LIN {X 0,Y 248.2,Z 586.565,A -85,B 0,C 180,E1 -18983.497,E2 -18983.497} C_VEL
LIN {X 0,Y 249.035,Z 580.902,A -85,B 0,C 180,E1 -18985.954,E2 -18985.954} C_VEL
LIN {X 0,Y 250.181,Z 573.816,A -85,B 0,C 180,E1 -18988.39,E2 -18988.39} C_VEL
LIN {X 0,Y 251.663,Z 564.939,A -85,B 0,C 180,E1 -18990.8,E2 -18990.8} C_VEL
LIN {X 0,Y 253.35,Z 554.938,A -85,B 0,C 180,E1 -18992.961,E2 -18992.961} C_VEL
LIN {X 0,Y 254.867,Z 544.511,A -85,B 0,C 180,E1 -18994.745,E2 -18994.745} C_VEL
LIN {X 0,Y 256.41,Z 533.043,A -85,B 0,C 180,E1 -18996.294,E2 -18996.294} C_VEL
LIN {X 0,Y 257.735,Z 521.099,A -85,B 0,C 180,E1 -18997.54,E2 -18997.54} C_VEL
LIN {X 0,Y 258.808,Z 507.869,A -85,B 0,C 180,E1 -18998.54,E2 -18998.54} C_VEL
LIN {X 0,Y 259.542,Z 494.726,A -85,B 0,C 180,E1 -18999.203,E2 -18999.203} C_VEL
LIN {X 0,Y 261.752,Z 423.09,A -85,B 0,C 180,E1 -19001.164,E2 -19001.164} C_VEL
LIN {X 0,Y 256.331,Z 407.243,A -85,B 0,C 180,E1 -19002.139,E2 -19002.139} C_VEL
LIN {X 0,Y 251.283,Z 395.565,A -85,B 0,C 180,E1 -19002.996,E2 -19002.996} C_VEL
LIN {X 0,Y 249.318,Z 390.908,A -85,B 0,C 180,E1 -19003.344,E2 -19003.344} C_VEL
LIN {X 0,Y 249.246,Z 390.443,A -85,B 0,C 180,E1 -19003.4,E2 -19003.4} C_VEL
LIN {X 0,Y 249.222,Z 390.442,A -85,B 0,C 180,E1 -19006.503,E2 -19006.503} C_VEL
LIN {X 0,Y 249.091,Z 390.458,A -85,B 0,C 180,E1 -19011.517,E2 -19011.517} C_VEL
LIN {X 0,Y 249.134,Z 390.45,A -85,B 0,C 180,E1 -19015.481,E2 -19015.481} C_VEL
LIN {X 0,Y 249.086,Z 390.458,A -85,B 0,C 180,E1 -19018.992,E2 -19018.992} C_VEL
LIN {X 0,Y 249.032,Z 390.462,A -85,B 0,C 180,E1 -19022.425,E2 -19022.425} C_VEL
LIN {X 0,Y 249.031,Z 390.461,A -85,B 0,C 180,E1 -19026.344,E2 -19026.344} C_VEL
LIN {X 0,Y 249.006,Z 390.465,A -85,B 0,C 180,E1 -19030.477,E2 -19030.477} C_VEL
LIN {X 0,Y 249.007,Z 390.468,A -85,B 0,C 180,E1 -19034.877,E2 -19034.877} C_VEL
LIN {X 0,Y 249.017,Z 390.463,A -85,B 0,C 180,E1 -19037.362,E2 -19037.362} C_VEL
LIN {X 0,Y 249.041,Z 390.458,A -85,B 0,C 180,E1 -19042.199,E2 -19042.199} C_VEL
LIN {X 0,Y 249.041,Z 390.462,A -85,B 0,C 180,E1 -19045.638,E2 -19045.638} C_VEL
LIN {X 0,Y 249.049,Z 390.456,A -85,B 0,C 180,E1 -19049.472,E2 -19049.472} C_VEL
LIN {X 0,Y 249.07,Z 390.459,A -85,B 0,C 180,E1 -19053.161,E2 -19053.161} C_VEL
LIN {X 0,Y 249.076,Z 390.454,A -85,B 0,C 180,E1 -19056.732,E2 -19056.732} C_VEL
LIN {X 0,Y 249.107,Z 390.453,A -85,B 0,C 180,E1 -19060.211,E2 -19060.211} C_VEL
LIN {X 0,Y 249.238,Z 390.43,A -85,B 0,C 180,E1 -19063.621,E2 -19063.621} C_VEL
LIN {X 0,Y 249.24,Z 390.437,A -85,B 0,C 180,E1 -19068.615,E2 -19068.615} C_VEL
LIN {X 0,Y 249.449,Z 390.406,A -85,B 0,C 180,E1 -19071.901,E2 -19071.901} C_VEL
LIN {X 0,Y 249.292,Z 390.429,A -85,B 0,C 180,E1 -19075.148,E2 -19075.148} C_VEL
LIN {X 0,Y 249.67,Z 390.375,A -85,B 0,C 180,E1 -19078.387,E2 -19078.387} C_VEL
LIN {X 0,Y 249.671,Z 390.358,A -85,B 0,C 180,E1 -19081.613,E2 -19081.613} C_VEL
LIN {X 0,Y 249.448,Z 390.411,A -85,B 0,C 180,E1 -19086.47,E2 -19086.47} C_VEL
LIN {X 0,Y 249.308,Z 390.425,A -85,B 0,C 180,E1 -19090.006,E2 -19090.006} C_VEL
LIN {X 0,Y 248.561,Z 390.517,A -85,B 0,C 180,E1 -19091.353,E2 -19091.353} C_VEL
LIN {X 0,Y 245.711,Z 390.875,A -85,B 0,C 180,E1 -19093.55,E2 -19093.55} C_VEL
LIN {X 0,Y 242.481,Z 391.281,A -85,B 0,C 180,E1 -19096.256,E2 -19096.256} C_VEL
LIN {X 0,Y 242.115,Z 391.32,A -85,B 0,C 180,E1 -19097.193,E2 -19097.193} C_VEL
LIN {X 0,Y 242.008,Z 391.34,A -85,B 0,C 180,E1 -19102.18,E2 -19102.18} C_VEL
LIN {X 0,Y 242.062,Z 391.333,A -85,B 0,C 180,E1 -19105.838,E2 -19105.838} C_VEL
LIN {X 0,Y 242.027,Z 391.337,A -85,B 0,C 180,E1 -19109.58,E2 -19109.58} C_VEL
LIN {X 0,Y 241.988,Z 391.343,A -85,B 0,C 180,E1 -19113.491,E2 -19113.491} C_VEL
LIN {X 0,Y 242.009,Z 391.342,A -85,B 0,C 180,E1 -19117.578,E2 -19117.578} C_VEL
LIN {X 0,Y 241.982,Z 391.348,A -85,B 0,C 180,E1 -19121.913,E2 -19121.913} C_VEL
LIN {X 0,Y 241.983,Z 391.344,A -85,B 0,C 180,E1 -19126.559,E2 -19126.559} C_VEL
LIN {X 0,Y 241.986,Z 391.339,A -85,B 0,C 180,E1 -19130.288,E2 -19130.288} C_VEL
LIN {X 0,Y 242.097,Z 391.377,A -85,B 0,C 180,E1 -19133.66,E2 -19133.66} C_VEL
LIN {X 0,Y 244.057,Z 400.843,A -85,B 0,C 180,E1 -19137.322,E2 -19137.322} C_VEL
LIN {X 0,Y 245.642,Z 408.584,A -85,B 0,C 180,E1 -19140.173,E2 -19140.173} C_VEL
LIN {X 0,Y 249.345,Z 419.538,A -85,B 0,C 180,E1 -19140.898,E2 -19140.898} C_VEL
LIN {X 0,Y 254.277,Z 461.944,A -85,B 0,C 180,E1 -19142.67,E2 -19142.67} C_VEL
LIN {X 0,Y 252.511,Z 517.102,A -85,B 0,C 180,E1 -19144.223,E2 -19144.223} C_VEL
LIN {X 0,Y 251.666,Z 530.452,A -85,B 0,C 180,E1 -19144.905,E2 -19144.905} C_VEL
LIN {X 0,Y 250.342,Z 543.226,A -85,B 0,C 180,E1 -19145.87,E2 -19145.87} C_VEL
LIN {X 0,Y 248.767,Z 555.378,A -85,B 0,C 180,E1 -19147.142,E2 -19147.142} C_VEL
LIN {X 0,Y 247.124,Z 565.64,A -85,B 0,C 180,E1 -19148.522,E2 -19148.522} C_VEL
LIN {X 0,Y 245.467,Z 576.326,A -85,B 0,C 180,E1 -19150.342,E2 -19150.342} C_VEL
LIN {X 0,Y 243.996,Z 584.587,A -85,B 0,C 180,E1 -19152.074,E2 -19152.074} C_VEL
LIN {X 0,Y 243.116,Z 590.805,A -85,B 0,C 180,E1 -19153.63,E2 -19153.63} C_VEL
LIN {X 0,Y 241.774,Z 599.073,A -85,B 0,C 180,E1 -19156.125,E2 -19156.125} C_VEL
LIN {X 0,Y 240.907,Z 604.686,A -85,B 0,C 180,E1 -19158.217,E2 -19158.217} C_VEL
LIN {X 0,Y 240.332,Z 610.169,A -85,B 0,C 180,E1 -19160.745,E2 -19160.745} C_VEL
LIN {X 0,Y 240.044,Z 614.433,A -85,B 0,C 180,E1 -19163.275,E2 -19163.275} C_VEL
LIN {X 0,Y 239.922,Z 616.68,A -85,B 0,C 180,E1 -19164.959,E2 -19164.959} C_VEL
LIN {X 0,Y 239.977,Z 618.439,A -85,B 0,C 180,E1 -19166.642,E2 -19166.642} C_VEL
LIN {X 0,Y 240.01,Z 619.761,A -85,B 0,C 180,E1 -19168.322,E2 -19168.322} C_VEL
LIN {X 0,Y 240.022,Z 620.676,A -85,B 0,C 180,E1 -19170,E2 -19170} C_VEL
LIN {X 0,Y 239.976,Z 621.188,A -85,B 0,C 180,E1 -19171.678,E2 -19171.678} C_VEL
LIN {X 0,Y 239.911,Z 621.261,A -85,B 0,C 180,E1 -19173.359,E2 -19173.359} C_VEL
LIN {X 0,Y 239.912,Z 620.913,A -85,B 0,C 180,E1 -19175.127,E2 -19175.127} C_VEL
LIN {X 0,Y 240.163,Z 619.15,A -85,B 0,C 180,E1 -19178.413,E2 -19178.413} C_VEL
LIN {X 0,Y 240.571,Z 617.639,A -85,B 0,C 180,E1 -19180.095,E2 -19180.095} C_VEL
LIN {X 0,Y 241.434,Z 614.593,A -85,B 0,C 180,E1 -19182.61,E2 -19182.61} C_VEL
LIN {X 0,Y 242.852,Z 610.525,A -85,B 0,C 180,E1 -19185.097,E2 -19185.097} C_VEL
LIN {X 0,Y 245.038,Z 604.321,A -85,B 0,C 180,E1 -19187.958,E2 -19187.958} C_VEL
LIN {X 0,Y 247.264,Z 597.853,A -85,B 0,C 180,E1 -19190.288,E2 -19190.288} C_VEL
LIN {X 0,Y 250.083,Z 589.313,A -85,B 0,C 180,E1 -19192.731,E2 -19192.731} C_VEL
LIN {X 0,Y 252.865,Z 580.828,A -85,B 0,C 180,E1 -19194.639,E2 -19194.639} C_VEL
LIN {X 0,Y 255.921,Z 570.39,A -85,B 0,C 180,E1 -19196.503,E2 -19196.503} C_VEL
LIN {X 0,Y 258.611,Z 560.094,A -85,B 0,C 180,E1 -19197.955,E2 -19197.955} C_VEL
LIN {X 0,Y 261.177,Z 548.836,A -85,B 0,C 180,E1 -19199.19,E2 -19199.19} C_VEL
LIN {X 0,Y 263.441,Z 536.133,A -85,B 0,C 180,E1 -19200.234,E2 -19200.234} C_VEL
LIN {X 0,Y 265.184,Z 522.682,A -85,B 0,C 180,E1 -19201.001,E2 -19201.001} C_VEL
LIN {X 0,Y 266.181,Z 510.056,A -85,B 0,C 180,E1 -19201.448,E2 -19201.448} C_VEL
LIN {X 0,Y 268.042,Z 465.142,A -85,B 0,C 180,E1 -19202.66,E2 -19202.66} C_VEL
LIN {X 0,Y 265.308,Z 446.292,A -85,B 0,C 180,E1 -19203.775,E2 -19203.775} C_VEL
LIN {X 0,Y 264.329,Z 441.703,A -85,B 0,C 180,E1 -19204.109,E2 -19204.109} C_VEL
LIN {X 0,Y 256.778,Z 425.571,A -85,B 0,C 180,E1 -19206.11,E2 -19206.11} C_VEL
LIN {X 0,Y 250.954,Z 414.885,A -85,B 0,C 180,E1 -19207.723,E2 -19207.723} C_VEL
LIN {X 0,Y 248.498,Z 410.557,A -85,B 0,C 180,E1 -19208.435,E2 -19208.435} C_VEL
LIN {X 0,Y 246.306,Z 406.343,A -85,B 0,C 180,E1 -19209.128,E2 -19209.128} C_VEL
LIN {X 0,Y 244.316,Z 399.158,A -85,B 0,C 180,E1 -19212.818,E2 -19212.818} C_VEL
LIN {X 0,Y 242.033,Z 391.332,A -85,B 0,C 180,E1 -19217.362,E2 -19217.362} C_VEL
LIN {X 0,Y 242.016,Z 391.34,A -85,B 0,C 180,E1 -19221.632,E2 -19221.632} C_VEL
LIN {X 0,Y 242.033,Z 391.336,A -85,B 0,C 180,E1 -19224.497,E2 -19224.497} C_VEL
LIN {X 0,Y 241.973,Z 391.343,A -85,B 0,C 180,E1 -19228.48,E2 -19228.48} C_VEL
LIN {X 0,Y 242.007,Z 391.338,A -85,B 0,C 180,E1 -19232.313,E2 -19232.313} C_VEL
LIN {X 0,Y 242.053,Z 391.334,A -85,B 0,C 180,E1 -19236.016,E2 -19236.016} C_VEL
LIN {X 0,Y 242.033,Z 391.331,A -85,B 0,C 180,E1 -19239.608,E2 -19239.608} C_VEL
LIN {X 0,Y 242.159,Z 391.308,A -85,B 0,C 180,E1 -19243.278,E2 -19243.278} C_VEL
LIN {X 0,Y 242.18,Z 391.306,A -85,B 0,C 180,E1 -19248.28,E2 -19248.28} C_VEL
LIN {X 0,Y 242.421,Z 391.276,A -85,B 0,C 180,E1 -19251.666,E2 -19251.666} C_VEL
LIN {X 0,Y 242.255,Z 391.309,A -85,B 0,C 180,E1 -19255.007,E2 -19255.007} C_VEL
LIN {X 0,Y 242.631,Z 391.25,A -85,B 0,C 180,E1 -19258.341,E2 -19258.341} C_VEL
LIN {X 0,Y 242.632,Z 391.25,A -85,B 0,C 180,E1 -19261.66,E2 -19261.66} C_VEL
LIN {X 0,Y 242.417,Z 391.277,A -85,B 0,C 180,E1 -19266.684,E2 -19266.684} C_VEL
LIN {X 0,Y 242.263,Z 391.308,A -85,B 0,C 180,E1 -19270.024,E2 -19270.024} C_VEL
LIN {X 0,Y 242.16,Z 391.315,A -85,B 0,C 180,E1 -19275.142,E2 -19275.142} C_VEL
LIN {X 0,Y 242.085,Z 391.331,A -85,B 0,C 180,E1 -19278.624,E2 -19278.624} C_VEL
LIN {X 0,Y 242.06,Z 391.334,A -85,B 0,C 180,E1 -19282.176,E2 -19282.176} C_VEL
LIN {X 0,Y 242.064,Z 391.333,A -85,B 0,C 180,E1 -19285.839,E2 -19285.839} C_VEL
LIN {X 0,Y 242.028,Z 391.335,A -85,B 0,C 180,E1 -19289.581,E2 -19289.581} C_VEL
LIN {X 0,Y 242.006,Z 391.394,A -85,B 0,C 180,E1 -19293.927,E2 -19293.927} C_VEL
LIN {X 0,Y 242.958,Z 394.034,A -85,B 0,C 180,E1 -19294.276,E2 -19294.276} C_VEL
LIN {X 0,Y 245.31,Z 396.811,A -85,B 0,C 180,E1 -19294.96,E2 -19294.96} C_VEL
LIN {X 0,Y 247.486,Z 400.114,A -85,B 0,C 180,E1 -19295.603,E2 -19295.603} C_VEL
LIN {X 0,Y 252.215,Z 407.1,A -85,B 0,C 180,E1 -19296.931,E2 -19296.931} C_VEL
LIN {X 0,Y 256.167,Z 413.341,A -85,B 0,C 180,E1 -19297.995,E2 -19297.995} C_VEL
LIN {X 0,Y 262.545,Z 425.008,A -85,B 0,C 180,E1 -19299.663,E2 -19299.663} C_VEL
LIN {X 0,Y 269.196,Z 439.033,A -85,B 0,C 180,E1 -19301.334,E2 -19301.334} C_VEL
LIN {X 0,Y 266.535,Z 496.566,A -85,B 0,C 180,E1 -19302.897,E2 -19302.897} C_VEL
LIN {X 0,Y 265.248,Z 510.053,A -85,B 0,C 180,E1 -19303.557,E2 -19303.557} C_VEL
LIN {X 0,Y 263.535,Z 522.714,A -85,B 0,C 180,E1 -19304.491,E2 -19304.491} C_VEL
LIN {X 0,Y 261.43,Z 534.297,A -85,B 0,C 180,E1 -19305.658,E2 -19305.658} C_VEL
LIN {X 0,Y 258.738,Z 546.27,A -85,B 0,C 180,E1 -19307.231,E2 -19307.231} C_VEL
LIN {X 0,Y 255.936,Z 556.885,A -85,B 0,C 180,E1 -19309.035,E2 -19309.035} C_VEL
LIN {X 0,Y 253.085,Z 566.205,A -85,B 0,C 180,E1 -19311.037,E2 -19311.037} C_VEL
LIN {X 0,Y 250.205,Z 574.762,A -85,B 0,C 180,E1 -19313.354,E2 -19313.354} C_VEL
LIN {X 0,Y 247.553,Z 582.051,A -85,B 0,C 180,E1 -19315.897,E2 -19315.897} C_VEL
LIN {X 0,Y 245.653,Z 586.942,A -85,B 0,C 180,E1 -19318.044,E2 -19318.044} C_VEL
LIN {X 0,Y 243.746,Z 591.546,A -85,B 0,C 180,E1 -19320.649,E2 -19320.649} C_VEL
LIN {X 0,Y 242.75,Z 593.944,A -85,B 0,C 180,E1 -19322.405,E2 -19322.405} C_VEL
LIN {X 0,Y 241.831,Z 595.977,A -85,B 0,C 180,E1 -19324.28,E2 -19324.28} C_VEL
LIN {X 0,Y 241.168,Z 597.278,A -85,B 0,C 180,E1 -19325.923,E2 -19325.923} C_VEL
LIN {X 0,Y 240.612,Z 598.253,A -85,B 0,C 180,E1 -19327.685,E2 -19327.685} C_VEL
LIN {X 0,Y 240.229,Z 598.811,A -85,B 0,C 180,E1 -19329.448,E2 -19329.448} C_VEL
LIN {X 0,Y 239.924,Z 598.91,A -85,B 0,C 180,E1 -19331.203,E2 -19331.203} C_VEL
LIN {X 0,Y 239.738,Z 598.584,A -85,B 0,C 180,E1 -19332.954,E2 -19332.954} C_VEL
LIN {X 0,Y 239.758,Z 597.487,A -85,B 0,C 180,E1 -19335.316,E2 -19335.316} C_VEL
LIN {X 0,Y 239.919,Z 595.083,A -85,B 0,C 180,E1 -19338.168,E2 -19338.168} C_VEL
LIN {X 0,Y 240.385,Z 591.842,A -85,B 0,C 180,E1 -19340.747,E2 -19340.747} C_VEL
LIN {X 0,Y 241.044,Z 587.519,A -85,B 0,C 180,E1 -19343.303,E2 -19343.303} C_VEL
LIN {X 0,Y 242.05,Z 580.982,A -85,B 0,C 180,E1 -19346.254,E2 -19346.254} C_VEL
LIN {X 0,Y 243.251,Z 573.809,A -85,B 0,C 180,E1 -19348.758,E2 -19348.758} C_VEL
LIN {X 0,Y 244.805,Z 564.86,A -85,B 0,C 180,E1 -19351.234,E2 -19351.234} C_VEL
LIN {X 0,Y 246.404,Z 555.67,A -85,B 0,C 180,E1 -19353.27,E2 -19353.27} C_VEL
LIN {X 0,Y 247.956,Z 545.486,A -85,B 0,C 180,E1 -19355.081,E2 -19355.081} C_VEL
LIN {X 0,Y 249.542,Z 534.158,A -85,B 0,C 180,E1 -19356.671,E2 -19356.671} C_VEL
LIN {X 0,Y 250.906,Z 522.441,A -85,B 0,C 180,E1 -19357.949,E2 -19357.949} C_VEL
LIN {X 0,Y 252.022,Z 509.688,A -85,B 0,C 180,E1 -19358.974,E2 -19358.974} C_VEL
LIN {X 0,Y 252.832,Z 496.157,A -85,B 0,C 180,E1 -19359.701,E2 -19359.701} C_VEL
LIN {X 0,Y 254.305,Z 452.666,A -85,B 0,C 180,E1 -19360.949,E2 -19360.949} C_VEL
LIN {X 0,Y 255.146,Z 424.433,A -85,B 0,C 180,E1 -19361.729,E2 -19361.729} C_VEL
LIN {X 0,Y 249.638,Z 408.47,A -85,B 0,C 180,E1 -19362.759,E2 -19362.759} C_VEL
LIN {X 0,Y 242.958,Z 393.784,A -85,B 0,C 180,E1 -19363.926,E2 -19363.926} C_VEL
LIN {X 0,Y 242.189,Z 391.321,A -85,B 0,C 180,E1 -19364.14,E2 -19364.14} C_VEL
LIN {X 0,Y 242.154,Z 391.324,A -85,B 0,C 180,E1 -19366.871,E2 -19366.871} C_VEL
LIN {X 0,Y 242.056,Z 391.333,A -85,B 0,C 180,E1 -19371.702,E2 -19371.702} C_VEL
LIN {X 0,Y 242.069,Z 391.332,A -85,B 0,C 180,E1 -19375.837,E2 -19375.837} C_VEL
LIN {X 0,Y 242.032,Z 391.338,A -85,B 0,C 180,E1 -19379.579,E2 -19379.579} C_VEL
LIN {X 0,Y 241.982,Z 391.344,A -85,B 0,C 180,E1 -19383.491,E2 -19383.491} C_VEL
LIN {X 0,Y 241.988,Z 391.34,A -85,B 0,C 180,E1 -19387.581,E2 -19387.581} C_VEL
LIN {X 0,Y 241.939,Z 391.342,A -85,B 0,C 180,E1 -19391.921,E2 -19391.921} C_VEL
LIN {X 0,Y 241.936,Z 391.344,A -85,B 0,C 180,E1 -19396.569,E2 -19396.569} C_VEL
LIN {X 0,Y 241.955,Z 391.344,A -85,B 0,C 180,E1 -19400.28,E2 -19400.28} C_VEL
LIN {X 0,Y 241.979,Z 391.34,A -85,B 0,C 180,E1 -19404.487,E2 -19404.487} C_VEL
LIN {X 0,Y 241.972,Z 391.342,A -85,B 0,C 180,E1 -19408.479,E2 -19408.479} C_VEL
LIN {X 0,Y 242.005,Z 391.338,A -85,B 0,C 180,E1 -19412.312,E2 -19412.312} C_VEL
LIN {X 0,Y 242.054,Z 391.327,A -85,B 0,C 180,E1 -19416.015,E2 -19416.015} C_VEL
LIN {X 0,Y 242.034,Z 391.334,A -85,B 0,C 180,E1 -19419.607,E2 -19419.607} C_VEL
LIN {X 0,Y 242.16,Z 391.312,A -85,B 0,C 180,E1 -19423.277,E2 -19423.277} C_VEL
LIN {X 0,Y 242.176,Z 391.317,A -85,B 0,C 180,E1 -19428.279,E2 -19428.279} C_VEL
LIN {X 0,Y 242.395,Z 391.284,A -85,B 0,C 180,E1 -19431.664,E2 -19431.664} C_VEL
LIN {X 0,Y 242.253,Z 391.306,A -85,B 0,C 180,E1 -19435.007,E2 -19435.007} C_VEL
LIN {X 0,Y 242.631,Z 391.251,A -85,B 0,C 180,E1 -19438.34,E2 -19438.34} C_VEL
LIN {X 0,Y 242.631,Z 391.233,A -85,B 0,C 180,E1 -19441.659,E2 -19441.659} C_VEL
LIN {X 0,Y 242.418,Z 391.288,A -85,B 0,C 180,E1 -19446.659,E2 -19446.659} C_VEL
LIN {X 0,Y 242.262,Z 391.307,A -85,B 0,C 180,E1 -19450.024,E2 -19450.024} C_VEL
LIN {X 0,Y 242.159,Z 391.319,A -85,B 0,C 180,E1 -19455.141,E2 -19455.141} C_VEL
LIN {X 0,Y 242.115,Z 391.32,A -85,B 0,C 180,E1 -19457.193,E2 -19457.193} C_VEL
LIN {X 0,Y 241.351,Z 391.419,A -85,B 0,C 180,E1 -19458.582,E2 -19458.582} C_VEL
LIN {X 0,Y 238.408,Z 391.787,A -85,B 0,C 180,E1 -19460.845,E2 -19460.845} C_VEL
LIN {X 0,Y 235.996,Z 392.085,A -85,B 0,C 180,E1 -19462.691,E2 -19462.691} C_VEL
LIN {X 0,Y 235.022,Z 392.207,A -85,B 0,C 180,E1 -19464.123,E2 -19464.123} C_VEL
LIN {X 0,Y 234.972,Z 392.214,A -85,B 0,C 180,E1 -19464.608,E2 -19464.608} C_VEL
LIN {X 0,Y 234.95,Z 392.219,A -85,B 0,C 180,E1 -19468.594,E2 -19468.594} C_VEL
LIN {X 0,Y 234.946,Z 392.22,A -85,B 0,C 180,E1 -19473.118,E2 -19473.118} C_VEL
LIN {X 0,Y 234.943,Z 392.222,A -85,B 0,C 180,E1 -19476.746,E2 -19476.746} C_VEL
LIN {X 0,Y 234.942,Z 392.223,A -85,B 0,C 180,E1 -19481.155,E2 -19481.155} C_VEL
LIN {X 0,Y 234.939,Z 392.224,A -85,B 0,C 180,E1 -19484.117,E2 -19484.117} C_VEL
LIN {X 0,Y 234.939,Z 392.22,A -85,B 0,C 180,E1 -19488.405,E2 -19488.405} C_VEL
LIN {X 0,Y 235.035,Z 392.347,A -85,B 0,C 180,E1 -19493.138,E2 -19493.138} C_VEL
LIN {X 0,Y 237.018,Z 401.538,A -85,B 0,C 180,E1 -19496.831,E2 -19496.831} C_VEL
LIN {X 0,Y 238.366,Z 408.281,A -85,B 0,C 180,E1 -19499.385,E2 -19499.385} C_VEL
LIN {X 0,Y 242.902,Z 420.907,A -85,B 0,C 180,E1 -19500.283,E2 -19500.283} C_VEL
LIN {X 0,Y 247.686,Z 462.997,A -85,B 0,C 180,E1 -19502.096,E2 -19502.096} C_VEL
LIN {X 0,Y 245.866,Z 516.715,A -85,B 0,C 180,E1 -19503.644,E2 -19503.644} C_VEL
LIN {X 0,Y 245.002,Z 530.089,A -85,B 0,C 180,E1 -19504.344,E2 -19504.344} C_VEL
LIN {X 0,Y 243.565,Z 543.426,A -85,B 0,C 180,E1 -19505.381,E2 -19505.381} C_VEL
LIN {X 0,Y 241.956,Z 555.431,A -85,B 0,C 180,E1 -19506.687,E2 -19506.687} C_VEL
LIN {X 0,Y 240.268,Z 565.623,A -85,B 0,C 180,E1 -19508.103,E2 -19508.103} C_VEL
LIN {X 0,Y 238.559,Z 576.255,A -85,B 0,C 180,E1 -19509.973,E2 -19509.973} C_VEL
LIN {X 0,Y 236.855,Z 586.018,A -85,B 0,C 180,E1 -19512.128,E2 -19512.128} C_VEL
LIN {X 0,Y 235.461,Z 594.309,A -85,B 0,C 180,E1 -19514.418,E2 -19514.418} C_VEL
LIN {X 0,Y 234.218,Z 601.815,A -85,B 0,C 180,E1 -19516.995,E2 -19516.995} C_VEL
LIN {X 0,Y 233.46,Z 607.834,A -85,B 0,C 180,E1 -19519.594,E2 -19519.594} C_VEL
LIN {X 0,Y 233.047,Z 612.567,A -85,B 0,C 180,E1 -19522.201,E2 -19522.201} C_VEL
LIN {X 0,Y 232.845,Z 616.267,A -85,B 0,C 180,E1 -19524.9,E2 -19524.9} C_VEL
LIN {X 0,Y 232.891,Z 617.97,A -85,B 0,C 180,E1 -19526.54,E2 -19526.54} C_VEL
LIN {X 0,Y 232.939,Z 619.324,A -85,B 0,C 180,E1 -19528.271,E2 -19528.271} C_VEL
LIN {X 0,Y 232.95,Z 620.268,A -85,B 0,C 180,E1 -19530,E2 -19530} C_VEL
LIN {X 0,Y 232.905,Z 620.812,A -85,B 0,C 180,E1 -19531.729,E2 -19531.729} C_VEL
LIN {X 0,Y 232.801,Z 620.715,A -85,B 0,C 180,E1 -19534.976,E2 -19534.976} C_VEL
LIN {X 0,Y 232.883,Z 619.974,A -85,B 0,C 180,E1 -19536.933,E2 -19536.933} C_VEL
LIN {X 0,Y 233.549,Z 617.467,A -85,B 0,C 180,E1 -19540.402,E2 -19540.402} C_VEL
LIN {X 0,Y 234.457,Z 614.472,A -85,B 0,C 180,E1 -19542.992,E2 -19542.992} C_VEL
LIN {X 0,Y 235.982,Z 610.466,A -85,B 0,C 180,E1 -19545.547,E2 -19545.547} C_VEL
LIN {X 0,Y 238.274,Z 604.363,A -85,B 0,C 180,E1 -19548.486,E2 -19548.486} C_VEL
LIN {X 0,Y 240.466,Z 598.409,A -85,B 0,C 180,E1 -19550.732,E2 -19550.732} C_VEL
LIN {X 0,Y 243.036,Z 591.024,A -85,B 0,C 180,E1 -19552.978,E2 -19552.978} C_VEL
LIN {X 0,Y 245.818,Z 582.974,A -85,B 0,C 180,E1 -19554.942,E2 -19554.942} C_VEL
LIN {X 0,Y 248.948,Z 573.186,A -85,B 0,C 180,E1 -19556.852,E2 -19556.852} C_VEL
LIN {X 0,Y 252.025,Z 562.289,A -85,B 0,C 180,E1 -19558.525,E2 -19558.525} C_VEL
LIN {X 0,Y 255.055,Z 549.886,A -85,B 0,C 180,E1 -19559.962,E2 -19559.962} C_VEL
LIN {X 0,Y 257.392,Z 537.756,A -85,B 0,C 180,E1 -19561.022,E2 -19561.022} C_VEL
LIN {X 0,Y 259.221,Z 525.047,A -85,B 0,C 180,E1 -19561.805,E2 -19561.805} C_VEL
LIN {X 0,Y 260.368,Z 512.937,A -85,B 0,C 180,E1 -19562.289,E2 -19562.289} C_VEL
LIN {X 0,Y 262.443,Z 466.155,A -85,B 0,C 180,E1 -19563.584,E2 -19563.584} C_VEL
LIN {X 0,Y 259.786,Z 447.749,A -85,B 0,C 180,E1 -19564.719,E2 -19564.719} C_VEL
LIN {X 0,Y 258.954,Z 444.374,A -85,B 0,C 180,E1 -19564.996,E2 -19564.996} C_VEL
LIN {X 0,Y 251.979,Z 429.485,A -85,B 0,C 180,E1 -19566.938,E2 -19566.938} C_VEL
LIN {X 0,Y 246.41,Z 418.994,A -85,B 0,C 180,E1 -19568.562,E2 -19568.562} C_VEL
LIN {X 0,Y 241.671,Z 410.659,A -85,B 0,C 180,E1 -19570.019,E2 -19570.019} C_VEL
LIN {X 0,Y 239.166,Z 406.342,A -85,B 0,C 180,E1 -19570.827,E2 -19570.827} C_VEL
LIN {X 0,Y 238.913,Z 405.628,A -85,B 0,C 180,E1 -19571.033,E2 -19571.033} C_VEL
LIN {X 0,Y 237.013,Z 399.189,A -85,B 0,C 180,E1 -19574.63,E2 -19574.63} C_VEL
LIN {X 0,Y 234.975,Z 392.217,A -85,B 0,C 180,E1 -19578.994,E2 -19578.994} C_VEL
LIN {X 0,Y 234.943,Z 392.212,A -85,B 0,C 180,E1 -19583.254,E2 -19583.254} C_VEL
LIN {X 0,Y 234.956,Z 392.212,A -85,B 0,C 180,E1 -19587.424,E2 -19587.424} C_VEL
LIN {X 0,Y 234.95,Z 392.215,A -85,B 0,C 180,E1 -19591.406,E2 -19591.406} C_VEL
LIN {X 0,Y 234.983,Z 392.209,A -85,B 0,C 180,E1 -19595.246,E2 -19595.246} C_VEL
LIN {X 0,Y 235.007,Z 392.201,A -85,B 0,C 180,E1 -19598.97,E2 -19598.97} C_VEL
LIN {X 0,Y 235.091,Z 392.187,A -85,B 0,C 180,E1 -19603.06,E2 -19603.06} C_VEL
LIN {X 0,Y 235.112,Z 392.185,A -85,B 0,C 180,E1 -19607.922,E2 -19607.922} C_VEL
LIN {X 0,Y 235.371,Z 392.156,A -85,B 0,C 180,E1 -19611.414,E2 -19611.414} C_VEL
LIN {X 0,Y 235.397,Z 392.148,A -85,B 0,C 180,E1 -19613.142,E2 -19613.142} C_VEL
LIN {X 0,Y 235.591,Z 392.126,A -85,B 0,C 180,E1 -19618.291,E2 -19618.291} C_VEL
LIN {X 0,Y 235.591,Z 392.126,A -85,B 0,C 180,E1 -19621.71,E2 -19621.71} C_VEL
LIN {X 0,Y 235.369,Z 392.154,A -85,B 0,C 180,E1 -19626.86,E2 -19626.86} C_VEL
LIN {X 0,Y 235.21,Z 392.185,A -85,B 0,C 180,E1 -19630.328,E2 -19630.328} C_VEL
LIN {X 0,Y 235.108,Z 392.189,A -85,B 0,C 180,E1 -19635.607,E2 -19635.607} C_VEL
LIN {X 0,Y 235.025,Z 392.205,A -85,B 0,C 180,E1 -19639.205,E2 -19639.205} C_VEL
LIN {X 0,Y 234.986,Z 392.21,A -85,B 0,C 180,E1 -19642.881,E2 -19642.881} C_VEL
LIN {X 0,Y 234.967,Z 392.212,A -85,B 0,C 180,E1 -19646.658,E2 -19646.658} C_VEL
LIN {X 0,Y 234.93,Z 392.216,A -85,B 0,C 180,E1 -19650.569,E2 -19650.569} C_VEL
LIN {X 0,Y 234.946,Z 392.219,A -85,B 0,C 180,E1 -19652.071,E2 -19652.071} C_VEL
LIN {X 0,Y 235.961,Z 395.087,A -85,B 0,C 180,E1 -19652.517,E2 -19652.517} C_VEL
LIN {X 0,Y 238.394,Z 397.754,A -85,B 0,C 180,E1 -19653.283,E2 -19653.283} C_VEL
LIN {X 0,Y 240.524,Z 401.042,A -85,B 0,C 180,E1 -19653.971,E2 -19653.971} C_VEL
LIN {X 0,Y 241.984,Z 402.995,A -85,B 0,C 180,E1 -19654.417,E2 -19654.417} C_VEL
LIN {X 0,Y 247.628,Z 411.237,A -85,B 0,C 180,E1 -19656.088,E2 -19656.088} C_VEL
LIN {X 0,Y 252.19,Z 418.616,A -85,B 0,C 180,E1 -19657.373,E2 -19657.373} C_VEL
LIN {X 0,Y 258.595,Z 430.57,A -85,B 0,C 180,E1 -19659.119,E2 -19659.119} C_VEL
LIN {X 0,Y 263.574,Z 441.238,A -85,B 0,C 180,E1 -19660.428,E2 -19660.428} C_VEL
LIN {X 0,Y 260.928,Z 496.621,A -85,B 0,C 180,E1 -19661.958,E2 -19661.958} C_VEL
LIN {X 0,Y 259.625,Z 509.957,A -85,B 0,C 180,E1 -19662.614,E2 -19662.614} C_VEL
LIN {X 0,Y 257.941,Z 522.004,A -85,B 0,C 180,E1 -19663.496,E2 -19663.496} C_VEL
LIN {X 0,Y 255.734,Z 533.877,A -85,B 0,C 180,E1 -19664.678,E2 -19664.678} C_VEL
LIN {X 0,Y 253.056,Z 545.623,A -85,B 0,C 180,E1 -19666.228,E2 -19666.228} C_VEL
LIN {X 0,Y 250.301,Z 555.665,A -85,B 0,C 180,E1 -19667.906,E2 -19667.906} C_VEL
LIN {X 0,Y 247.333,Z 565.115,A -85,B 0,C 180,E1 -19669.897,E2 -19669.897} C_VEL
LIN {X 0,Y 244.2,Z 574.052,A -85,B 0,C 180,E1 -19672.298,E2 -19672.298} C_VEL
LIN {X 0,Y 241.277,Z 581.709,A -85,B 0,C 180,E1 -19674.934,E2 -19674.934} C_VEL
LIN {X 0,Y 239.284,Z 586.61,A -85,B 0,C 180,E1 -19677.088,E2 -19677.088} C_VEL
LIN {X 0,Y 237.219,Z 591.397,A -85,B 0,C 180,E1 -19679.759,E2 -19679.759} C_VEL
LIN {X 0,Y 235.593,Z 594.954,A -85,B 0,C 180,E1 -19682.46,E2 -19682.46} C_VEL
LIN {X 0,Y 234.344,Z 597.405,A -85,B 0,C 180,E1 -19685.175,E2 -19685.175} C_VEL
LIN {X 0,Y 233.719,Z 598.443,A -85,B 0,C 180,E1 -19686.989,E2 -19686.989} C_VEL
LIN {X 0,Y 233.218,Z 599.137,A -85,B 0,C 180,E1 -19689.098,E2 -19689.098} C_VEL
LIN {X 0,Y 232.704,Z 599.019,A -85,B 0,C 180,E1 -19692.422,E2 -19692.422} C_VEL
LIN {X 0,Y 232.661,Z 597.845,A -85,B 0,C 180,E1 -19695.159,E2 -19695.159} C_VEL
LIN {X 0,Y 232.797,Z 595.763,A -85,B 0,C 180,E1 -19697.8,E2 -19697.8} C_VEL
LIN {X 0,Y 233.228,Z 592.651,A -85,B 0,C 180,E1 -19700.46,E2 -19700.46} C_VEL
LIN {X 0,Y 233.881,Z 588.463,A -85,B 0,C 180,E1 -19703.097,E2 -19703.097} C_VEL
LIN {X 0,Y 234.895,Z 582.072,A -85,B 0,C 180,E1 -19706.14,E2 -19706.14} C_VEL
LIN {X 0,Y 236.112,Z 575.12,A -85,B 0,C 180,E1 -19708.721,E2 -19708.721} C_VEL
LIN {X 0,Y 237.661,Z 566.409,A -85,B 0,C 180,E1 -19711.271,E2 -19711.271} C_VEL
LIN {X 0,Y 239.411,Z 556.66,A -85,B 0,C 180,E1 -19713.537,E2 -19713.537} C_VEL
LIN {X 0,Y 241.055,Z 546.44,A -85,B 0,C 180,E1 -19715.437,E2 -19715.437} C_VEL
LIN {X 0,Y 242.683,Z 535.256,A -85,B 0,C 180,E1 -19717.07,E2 -19717.07} C_VEL
LIN {X 0,Y 244.209,Z 522.736,A -85,B 0,C 180,E1 -19718.481,E2 -19718.481} C_VEL
LIN {X 0,Y 245.351,Z 509.978,A -85,B 0,C 180,E1 -19719.532,E2 -19719.532} C_VEL
LIN {X 0,Y 246.213,Z 496.07,A -85,B 0,C 180,E1 -19720.292,E2 -19720.292} C_VEL
LIN {X 0,Y 248.548,Z 425.66,A -85,B 0,C 180,E1 -19722.329,E2 -19722.329} C_VEL
LIN {X 0,Y 243.034,Z 409.951,A -85,B 0,C 180,E1 -19723.395,E2 -19723.395} C_VEL
LIN {X 0,Y 235.305,Z 393.123,A -85,B 0,C 180,E1 -19724.806,E2 -19724.806} C_VEL
LIN {X 0,Y 235.14,Z 392.199,A -85,B 0,C 180,E1 -19724.879,E2 -19724.879} C_VEL
LIN {X 0,Y 235.013,Z 392.213,A -85,B 0,C 180,E1 -19729.205,E2 -19729.205} C_VEL
LIN {X 0,Y 234.964,Z 392.213,A -85,B 0,C 180,E1 -19732.882,E2 -19732.882} C_VEL
LIN {X 0,Y 234.973,Z 392.216,A -85,B 0,C 180,E1 -19736.656,E2 -19736.656} C_VEL
LIN {X 0,Y 234.934,Z 392.221,A -85,B 0,C 180,E1 -19740.567,E2 -19740.567} C_VEL
LIN {X 0,Y 234.928,Z 392.221,A -85,B 0,C 180,E1 -19744.637,E2 -19744.637} C_VEL
LIN {X 0,Y 234.942,Z 392.22,A -85,B 0,C 180,E1 -19748.943,E2 -19748.943} C_VEL
LIN {X 0,Y 234.889,Z 392.225,A -85,B 0,C 180,E1 -19753.484,E2 -19753.484} C_VEL
LIN {X 0,Y 234.889,Z 392.222,A -85,B 0,C 180,E1 -19756.513,E2 -19756.513} C_VEL
LIN {X 0,Y 234.917,Z 392.22,A -85,B 0,C 180,E1 -19761.078,E2 -19761.078} C_VEL
LIN {X 0,Y 234.924,Z 392.221,A -85,B 0,C 180,E1 -19765.36,E2 -19765.36} C_VEL
LIN {X 0,Y 234.929,Z 392.215,A -85,B 0,C 180,E1 -19769.431,E2 -19769.431} C_VEL
LIN {X 0,Y 234.991,Z 392.211,A -85,B 0,C 180,E1 -19773.793,E2 -19773.793} C_VEL
LIN {X 0,Y 235.008,Z 392.211,A -85,B 0,C 180,E1 -19778.969,E2 -19778.969} C_VEL
LIN {X 0,Y 235.093,Z 392.193,A -85,B 0,C 180,E1 -19783.059,E2 -19783.059} C_VEL
LIN {X 0,Y 235.11,Z 392.196,A -85,B 0,C 180,E1 -19787.921,E2 -19787.921} C_VEL
LIN {X 0,Y 235.326,Z 392.164,A -85,B 0,C 180,E1 -19791.412,E2 -19791.412} C_VEL
LIN {X 0,Y 235.388,Z 392.161,A -85,B 0,C 180,E1 -19793.14,E2 -19793.14} C_VEL
LIN {X 0,Y 235.591,Z 392.128,A -85,B 0,C 180,E1 -19798.29,E2 -19798.29} C_VEL
LIN {X 0,Y 235.591,Z 392.109,A -85,B 0,C 180,E1 -19801.709,E2 -19801.709} C_VEL
LIN {X 0,Y 235.368,Z 392.165,A -85,B 0,C 180,E1 -19806.859,E2 -19806.859} C_VEL
LIN {X 0,Y 235.209,Z 392.184,A -85,B 0,C 180,E1 -19810.327,E2 -19810.327} C_VEL
LIN {X 0,Y 235.107,Z 392.198,A -85,B 0,C 180,E1 -19815.607,E2 -19815.607} C_VEL
LIN {X 0,Y 235.004,Z 392.208,A -85,B 0,C 180,E1 -19819.206,E2 -19819.206} C_VEL
LIN {X 0,Y 234.956,Z 392.214,A -85,B 0,C 180,E1 -19822.883,E2 -19822.883} C_VEL
LIN {X 0,Y 234.972,Z 392.214,A -85,B 0,C 180,E1 -19824.608,E2 -19824.608} C_VEL
LIN {X 0,Y 234.71,Z 392.254,A -85,B 0,C 180,E1 -19825.566,E2 -19825.566} C_VEL
LIN {X 0,Y 233.395,Z 392.423,A -85,B 0,C 180,E1 -19826.98,E2 -19826.98} C_VEL
LIN {X 0,Y 229.017,Z 392.962,A -85,B 0,C 180,E1 -19830.277,E2 -19830.277} C_VEL
LIN {X 0,Y 227.936,Z 393.093,A -85,B 0,C 180,E1 -19831.756,E2 -19831.756} C_VEL
LIN {X 0,Y 227.845,Z 393.101,A -85,B 0,C 180,E1 -19832.259,E2 -19832.259} C_VEL
LIN {X 0,Y 227.905,Z 393.1,A -85,B 0,C 180,E1 -19836.702,E2 -19836.702} C_VEL
LIN {X 0,Y 227.889,Z 393.104,A -85,B 0,C 180,E1 -19840.363,E2 -19840.363} C_VEL
LIN {X 0,Y 227.907,Z 393.099,A -85,B 0,C 180,E1 -19842.72,E2 -19842.72} C_VEL
LIN {X 0,Y 227.896,Z 393.099,A -85,B 0,C 180,E1 -19847.742,E2 -19847.742} C_VEL
LIN {X 0,Y 227.991,Z 393.185,A -85,B 0,C 180,E1 -19852.533,E2 -19852.533} C_VEL
LIN {X 0,Y 230.102,Z 403.073,A -85,B 0,C 180,E1 -19856.649,E2 -19856.649} C_VEL
LIN {X 0,Y 231.12,Z 408.028,A -85,B 0,C 180,E1 -19858.551,E2 -19858.551} C_VEL
LIN {X 0,Y 236.559,Z 423.076,A -85,B 0,C 180,E1 -19859.677,E2 -19859.677} C_VEL
LIN {X 0,Y 241.104,Z 462.922,A -85,B 0,C 180,E1 -19861.455,E2 -19861.455} C_VEL
LIN {X 0,Y 239.277,Z 516.346,A -85,B 0,C 180,E1 -19863.037,E2 -19863.037} C_VEL
LIN {X 0,Y 238.359,Z 529.724,A -85,B 0,C 180,E1 -19863.752,E2 -19863.752} C_VEL
LIN {X 0,Y 236.98,Z 542.524,A -85,B 0,C 180,E1 -19864.767,E2 -19864.767} C_VEL
LIN {X 0,Y 235.424,Z 553.89,A -85,B 0,C 180,E1 -19866,E2 -19866} C_VEL
LIN {X 0,Y 233.424,Z 565.606,A -85,B 0,C 180,E1 -19867.66,E2 -19867.66} C_VEL
LIN {X 0,Y 231.659,Z 576.185,A -85,B 0,C 180,E1 -19869.581,E2 -19869.581} C_VEL
LIN {X 0,Y 229.865,Z 586.001,A -85,B 0,C 180,E1 -19871.829,E2 -19871.829} C_VEL
LIN {X 0,Y 228.55,Z 593.451,A -85,B 0,C 180,E1 -19873.934,E2 -19873.934} C_VEL
LIN {X 0,Y 227.27,Z 601.054,A -85,B 0,C 180,E1 -19876.59,E2 -19876.59} C_VEL
LIN {X 0,Y 226.448,Z 607.153,A -85,B 0,C 180,E1 -19879.268,E2 -19879.268} C_VEL
LIN {X 0,Y 226.002,Z 611.961,A -85,B 0,C 180,E1 -19881.956,E2 -19881.956} C_VEL
LIN {X 0,Y 225.751,Z 616.051,A -85,B 0,C 180,E1 -19885.01,E2 -19885.01} C_VEL
LIN {X 0,Y 225.868,Z 618.884,A -85,B 0,C 180,E1 -19888.217,E2 -19888.217} C_VEL
LIN {X 0,Y 225.879,Z 619.859,A -85,B 0,C 180,E1 -19890,E2 -19890} C_VEL
LIN {X 0,Y 225.833,Z 620.433,A -85,B 0,C 180,E1 -19891.783,E2 -19891.783} C_VEL
LIN {X 0,Y 225.723,Z 620.462,A -85,B 0,C 180,E1 -19894.906,E2 -19894.906} C_VEL
LIN {X 0,Y 225.811,Z 619.713,A -85,B 0,C 180,E1 -19897.151,E2 -19897.151} C_VEL
LIN {X 0,Y 226.544,Z 617.277,A -85,B 0,C 180,E1 -19900.727,E2 -19900.727} C_VEL
LIN {X 0,Y 227.505,Z 614.336,A -85,B 0,C 180,E1 -19903.396,E2 -19903.396} C_VEL
LIN {X 0,Y 229.134,Z 610.401,A -85,B 0,C 180,E1 -19906.024,E2 -19906.024} C_VEL
LIN {X 0,Y 231.16,Z 605.367,A -85,B 0,C 180,E1 -19908.616,E2 -19908.616} C_VEL
LIN {X 0,Y 233.62,Z 599.086,A -85,B 0,C 180,E1 -19911.161,E2 -19911.161} C_VEL
LIN {X 0,Y 236.524,Z 591.274,A -85,B 0,C 180,E1 -19913.649,E2 -19913.649} C_VEL
LIN {X 0,Y 239.412,Z 583.34,A -85,B 0,C 180,E1 -19915.657,E2 -19915.657} C_VEL
LIN {X 0,Y 243.015,Z 572.626,A -85,B 0,C 180,E1 -19917.796,E2 -19917.796} C_VEL
LIN {X 0,Y 246.253,Z 561.653,A -85,B 0,C 180,E1 -19919.492,E2 -19919.492} C_VEL
LIN {X 0,Y 249.354,Z 549.187,A -85,B 0,C 180,E1 -19920.955,E2 -19920.955} C_VEL
LIN {X 0,Y 251.812,Z 536.935,A -85,B 0,C 180,E1 -19922.024,E2 -19922.024} C_VEL
LIN {X 0,Y 253.681,Z 524.023,A -85,B 0,C 180,E1 -19922.816,E2 -19922.816} C_VEL
LIN {X 0,Y 254.929,Z 510.4,A -85,B 0,C 180,E1 -19923.342,E2 -19923.342} C_VEL
LIN {X 0,Y 256.895,Z 467.248,A -85,B 0,C 180,E1 -19924.55,E2 -19924.55} C_VEL
LIN {X 0,Y 254.364,Z 449.155,A -85,B 0,C 180,E1 -19925.704,E2 -19925.704} C_VEL
LIN {X 0,Y 250.536,Z 440.152,A -85,B 0,C 180,E1 -19926.826,E2 -19926.826} C_VEL
LIN {X 0,Y 245.169,Z 429.269,A -85,B 0,C 180,E1 -19928.423,E2 -19928.423} C_VEL
LIN {X 0,Y 240.012,Z 419.783,A -85,B 0,C 180,E1 -19930.035,E2 -19930.035} C_VEL
LIN {X 0,Y 237.21,Z 414.889,A -85,B 0,C 180,E1 -19930.953,E2 -19930.953} C_VEL
LIN {X 0,Y 234.532,Z 410.337,A -85,B 0,C 180,E1 -19931.86,E2 -19931.86} C_VEL
LIN {X 0,Y 231.969,Z 406.29,A -85,B 0,C 180,E1 -19932.756,E2 -19932.756} C_VEL
LIN {X 0,Y 231.55,Z 405.278,A -85,B 0,C 180,E1 -19932.978,E2 -19932.978} C_VEL
LIN {X 0,Y 229.292,Z 397.671,A -85,B 0,C 180,E1 -19937.599,E2 -19937.599} C_VEL
LIN {X 0,Y 227.914,Z 393.09,A -85,B 0,C 180,E1 -19940.782,E2 -19940.782} C_VEL
LIN {X 0,Y 227.898,Z 393.093,A -85,B 0,C 180,E1 -19944.132,E2 -19944.132} C_VEL
LIN {X 0,Y 227.869,Z 393.1,A -85,B 0,C 180,E1 -19948.378,E2 -19948.378} C_VEL
LIN {X 0,Y 227.884,Z 393.096,A -85,B 0,C 180,E1 -19952.445,E2 -19952.445} C_VEL
LIN {X 0,Y 227.91,Z 393.095,A -85,B 0,C 180,E1 -19956.367,E2 -19956.367} C_VEL
LIN {X 0,Y 227.937,Z 393.093,A -85,B 0,C 180,E1 -19960.174,E2 -19960.174} C_VEL
LIN {X 0,Y 228.049,Z 393.069,A -85,B 0,C 180,E1 -19963.898,E2 -19963.898} C_VEL
LIN {X 0,Y 228.068,Z 393.061,A -85,B 0,C 180,E1 -19967.543,E2 -19967.543} C_VEL
LIN {X 0,Y 228.3,Z 393.039,A -85,B 0,C 180,E1 -19971.146,E2 -19971.146} C_VEL
LIN {X 0,Y 228.348,Z 393.025,A -85,B 0,C 180,E1 -19972.929,E2 -19972.929} C_VEL
LIN {X 0,Y 228.55,Z 393.002,A -85,B 0,C 180,E1 -19978.238,E2 -19978.238} C_VEL
LIN {X 0,Y 228.55,Z 393.003,A -85,B 0,C 180,E1 -19981.763,E2 -19981.763} C_VEL
LIN {X 0,Y 228.32,Z 393.031,A -85,B 0,C 180,E1 -19987.073,E2 -19987.073} C_VEL
LIN {X 0,Y 228.141,Z 393.061,A -85,B 0,C 180,E1 -19990.652,E2 -19990.652} C_VEL
LIN {X 0,Y 228.059,Z 393.078,A -85,B 0,C 180,E1 -19994.273,E2 -19994.273} C_VEL
LIN {X 0,Y 228.007,Z 393.083,A -85,B 0,C 180,E1 -19997.954,E2 -19997.954} C_VEL
LIN {X 0,Y 227.97,Z 393.089,A -85,B 0,C 180,E1 -20002.356,E2 -20002.356} C_VEL
LIN {X 0,Y 227.94,Z 393.087,A -85,B 0,C 180,E1 -20006.604,E2 -20006.604} C_VEL
LIN {X 0,Y 227.904,Z 393.091,A -85,B 0,C 180,E1 -20010.096,E2 -20010.096} C_VEL
LIN {X 0,Y 228.8,Z 395.764,A -85,B 0,C 180,E1 -20010.504,E2 -20010.504} C_VEL
LIN {X 0,Y 230.744,Z 397.934,A -85,B 0,C 180,E1 -20011.185,E2 -20011.185} C_VEL
LIN {X 0,Y 231.519,Z 398.801,A -85,B 0,C 180,E1 -20011.45,E2 -20011.45} C_VEL
LIN {X 0,Y 233.655,Z 402.058,A -85,B 0,C 180,E1 -20012.206,E2 -20012.206} C_VEL
LIN {X 0,Y 235.129,Z 403.887,A -85,B 0,C 180,E1 -20012.694,E2 -20012.694} C_VEL
LIN {X 0,Y 241.26,Z 412.675,A -85,B 0,C 180,E1 -20014.652,E2 -20014.652} C_VEL
LIN {X 0,Y 247.229,Z 421.984,A -85,B 0,C 180,E1 -20016.432,E2 -20016.432} C_VEL
LIN {X 0,Y 253.947,Z 434.745,A -85,B 0,C 180,E1 -20018.355,E2 -20018.355} C_VEL
LIN {X 0,Y 258.06,Z 443.736,A -85,B 0,C 180,E1 -20019.5,E2 -20019.5} C_VEL
LIN {X 0,Y 255.345,Z 497.015,A -85,B 0,C 180,E1 -20020.988,E2 -20020.988} C_VEL
LIN {X 0,Y 253.988,Z 510.445,A -85,B 0,C 180,E1 -20021.661,E2 -20021.661} C_VEL
LIN {X 0,Y 252.231,Z 522.454,A -85,B 0,C 180,E1 -20022.556,E2 -20022.556} C_VEL
LIN {X 0,Y 250.133,Z 533.45,A -85,B 0,C 180,E1 -20023.657,E2 -20023.657} C_VEL
LIN {X 0,Y 247.57,Z 544.398,A -85,B 0,C 180,E1 -20025.086,E2 -20025.086} C_VEL
LIN {X 0,Y 244.73,Z 554.357,A -85,B 0,C 180,E1 -20026.716,E2 -20026.716} C_VEL
LIN {X 0,Y 241.409,Z 564.808,A -85,B 0,C 180,E1 -20028.9,E2 -20028.9} C_VEL
LIN {X 0,Y 238.287,Z 573.358,A -85,B 0,C 180,E1 -20031.191,E2 -20031.191} C_VEL
LIN {X 0,Y 235.259,Z 580.913,A -85,B 0,C 180,E1 -20033.764,E2 -20033.764} C_VEL
LIN {X 0,Y 232.989,Z 586.262,A -85,B 0,C 180,E1 -20036.08,E2 -20036.08} C_VEL
LIN {X 0,Y 230.727,Z 591.199,A -85,B 0,C 180,E1 -20038.814,E2 -20038.814} C_VEL
LIN {X 0,Y 228.961,Z 594.903,A -85,B 0,C 180,E1 -20041.591,E2 -20041.591} C_VEL
LIN {X 0,Y 227.564,Z 597.485,A -85,B 0,C 180,E1 -20044.383,E2 -20044.383} C_VEL
LIN {X 0,Y 226.862,Z 598.634,A -85,B 0,C 180,E1 -20046.252,E2 -20046.252} C_VEL
LIN {X 0,Y 226.179,Z 599.478,A -85,B 0,C 180,E1 -20048.78,E2 -20048.78} C_VEL
LIN {X 0,Y 225.658,Z 599.452,A -85,B 0,C 180,E1 -20051.854,E2 -20051.854} C_VEL
LIN {X 0,Y 225.576,Z 598.209,A -85,B 0,C 180,E1 -20054.982,E2 -20054.982} C_VEL
LIN {X 0,Y 225.665,Z 596.418,A -85,B 0,C 180,E1 -20057.408,E2 -20057.408} C_VEL
LIN {X 0,Y 226.069,Z 593.429,A -85,B 0,C 180,E1 -20060.155,E2 -20060.155} C_VEL
LIN {X 0,Y 226.737,Z 589.382,A -85,B 0,C 180,E1 -20062.878,E2 -20062.878} C_VEL
LIN {X 0,Y 227.718,Z 583.166,A -85,B 0,C 180,E1 -20066.018,E2 -20066.018} C_VEL
LIN {X 0,Y 228.925,Z 576.381,A -85,B 0,C 180,E1 -20068.681,E2 -20068.681} C_VEL
LIN {X 0,Y 230.532,Z 567.949,A -85,B 0,C 180,E1 -20071.31,E2 -20071.31} C_VEL
LIN {X 0,Y 232.149,Z 559.248,A -85,B 0,C 180,E1 -20073.471,E2 -20073.471} C_VEL
LIN {X 0,Y 233.989,Z 548.537,A -85,B 0,C 180,E1 -20075.602,E2 -20075.602} C_VEL
LIN {X 0,Y 235.609,Z 537.901,A -85,B 0,C 180,E1 -20077.283,E2 -20077.283} C_VEL
LIN {X 0,Y 237.194,Z 526.011,A -85,B 0,C 180,E1 -20078.734,E2 -20078.734} C_VEL
LIN {X 0,Y 238.474,Z 513.67,A -85,B 0,C 180,E1 -20079.863,E2 -20079.863} C_VEL
LIN {X 0,Y 239.383,Z 501.12,A -85,B 0,C 180,E1 -20080.676,E2 -20080.676} C_VEL
LIN {X 0,Y 239.995,Z 486.52,A -85,B 0,C 180,E1 -20081.232,E2 -20081.232} C_VEL
LIN {X 0,Y 242.003,Z 426.987,A -85,B 0,C 180,E1 -20082.953,E2 -20082.953} C_VEL
LIN {X 0,Y 236.941,Z 412.801,A -85,B 0,C 180,E1 -20083.961,E2 -20083.961} C_VEL
LIN {X 0,Y 229.055,Z 395.89,A -85,B 0,C 180,E1 -20085.458,E2 -20085.458} C_VEL
LIN {X 0,Y 228.082,Z 393.077,A -85,B 0,C 180,E1 -20085.693,E2 -20085.693} C_VEL
LIN {X 0,Y 227.946,Z 393.092,A -85,B 0,C 180,E1 -20089.825,E2 -20089.825} C_VEL
LIN {X 0,Y 227.917,Z 393.084,A -85,B 0,C 180,E1 -20093.632,E2 -20093.632} C_VEL
LIN {X 0,Y 227.889,Z 393.099,A -85,B 0,C 180,E1 -20097.554,E2 -20097.554} C_VEL
LIN {X 0,Y 227.872,Z 393.099,A -85,B 0,C 180,E1 -20101.621,E2 -20101.621} C_VEL
LIN {X 0,Y 227.881,Z 393.096,A -85,B 0,C 180,E1 -20105.871,E2 -20105.871} C_VEL
LIN {X 0,Y 227.827,Z 393.103,A -85,B 0,C 180,E1 -20110.375,E2 -20110.375} C_VEL
LIN {X 0,Y 227.835,Z 393.102,A -85,B 0,C 180,E1 -20115.191,E2 -20115.191} C_VEL
LIN {X 0,Y 227.825,Z 393.104,A -85,B 0,C 180,E1 -20119.622,E2 -20119.622} C_VEL
LIN {X 0,Y 227.878,Z 393.095,A -85,B 0,C 180,E1 -20124.127,E2 -20124.127} C_VEL
LIN {X 0,Y 227.868,Z 393.098,A -85,B 0,C 180,E1 -20128.377,E2 -20128.377} C_VEL
LIN {X 0,Y 227.883,Z 393.098,A -85,B 0,C 180,E1 -20132.444,E2 -20132.444} C_VEL
LIN {X 0,Y 227.911,Z 393.089,A -85,B 0,C 180,E1 -20136.366,E2 -20136.366} C_VEL
LIN {X 0,Y 227.939,Z 393.09,A -85,B 0,C 180,E1 -20140.174,E2 -20140.174} C_VEL
LIN {X 0,Y 228.054,Z 393.068,A -85,B 0,C 180,E1 -20143.897,E2 -20143.897} C_VEL
LIN {X 0,Y 228.068,Z 393.073,A -85,B 0,C 180,E1 -20147.542,E2 -20147.542} C_VEL
LIN {X 0,Y 228.263,Z 393.045,A -85,B 0,C 180,E1 -20151.144,E2 -20151.144} C_VEL
LIN {X 0,Y 228.335,Z 393.041,A -85,B 0,C 180,E1 -20152.927,E2 -20152.927} C_VEL
LIN {X 0,Y 228.549,Z 393.004,A -85,B 0,C 180,E1 -20158.237,E2 -20158.237} C_VEL
LIN {X 0,Y 228.549,Z 392.984,A -85,B 0,C 180,E1 -20161.762,E2 -20161.762} C_VEL
LIN {X 0,Y 228.319,Z 393.043,A -85,B 0,C 180,E1 -20167.072,E2 -20167.072} C_VEL
LIN {X 0,Y 228.141,Z 393.062,A -85,B 0,C 180,E1 -20170.651,E2 -20170.651} C_VEL
LIN {X 0,Y 228.058,Z 393.077,A -85,B 0,C 180,E1 -20174.272,E2 -20174.272} C_VEL
LIN {X 0,Y 227.999,Z 393.08,A -85,B 0,C 180,E1 -20177.953,E2 -20177.953} C_VEL
LIN {X 0,Y 227.926,Z 393.092,A -85,B 0,C 180,E1 -20182.329,E2 -20182.329} C_VEL
LIN {X 0,Y 227.939,Z 393.091,A -85,B 0,C 180,E1 -20186.603,E2 -20186.603} C_VEL
LIN {X 0,Y 227.905,Z 393.099,A -85,B 0,C 180,E1 -20190.297,E2 -20190.297} C_VEL
LIN {X 0,Y 227.845,Z 393.101,A -85,B 0,C 180,E1 -20192.259,E2 -20192.259} C_VEL
LIN {X 0,Y 227.169,Z 393.191,A -85,B 0,C 180,E1 -20193.735,E2 -20193.735} C_VEL
LIN {X 0,Y 224.33,Z 393.544,A -85,B 0,C 180,E1 -20196.145,E2 -20196.145} C_VEL
LIN {X 0,Y 221.934,Z 393.846,A -85,B 0,C 180,E1 -20198.111,E2 -20198.111} C_VEL
LIN {X 0,Y 220.922,Z 393.971,A -85,B 0,C 180,E1 -20199.637,E2 -20199.637} C_VEL
LIN {X 0,Y 220.848,Z 393.981,A -85,B 0,C 180,E1 -20200.154,E2 -20200.154} C_VEL
LIN {X 0,Y 220.83,Z 393.981,A -85,B 0,C 180,E1 -20204.439,E2 -20204.439} C_VEL
LIN {X 0,Y 220.841,Z 393.978,A -85,B 0,C 180,E1 -20208.065,E2 -20208.065} C_VEL
LIN {X 0,Y 220.922,Z 394.143,A -85,B 0,C 180,E1 -20211.943,E2 -20211.943} C_VEL
LIN {X 0,Y 223.002,Z 403.475,A -85,B 0,C 180,E1 -20215.987,E2 -20215.987} C_VEL
LIN {X 0,Y 223.751,Z 407.455,A -85,B 0,C 180,E1 -20217.629,E2 -20217.629} C_VEL
LIN {X 0,Y 230.228,Z 424.97,A -85,B 0,C 180,E1 -20219.028,E2 -20219.028} C_VEL
LIN {X 0,Y 234.548,Z 464.038,A -85,B 0,C 180,E1 -20220.823,E2 -20220.823} C_VEL
LIN {X 0,Y 232.661,Z 516.438,A -85,B 0,C 180,E1 -20222.416,E2 -20222.416} C_VEL
LIN {X 0,Y 231.671,Z 530.094,A -85,B 0,C 180,E1 -20223.177,E2 -20223.177} C_VEL
LIN {X 0,Y 230.251,Z 542.71,A -85,B 0,C 180,E1 -20224.218,E2 -20224.218} C_VEL
LIN {X 0,Y 228.654,Z 553.933,A -85,B 0,C 180,E1 -20225.485,E2 -20225.485} C_VEL
LIN {X 0,Y 226.595,Z 565.583,A -85,B 0,C 180,E1 -20227.189,E2 -20227.189} C_VEL
LIN {X 0,Y 224.771,Z 576.113,A -85,B 0,C 180,E1 -20229.166,E2 -20229.166} C_VEL
LIN {X 0,Y 223.039,Z 584.621,A -85,B 0,C 180,E1 -20231.142,E2 -20231.142} C_VEL
LIN {X 0,Y 221.989,Z 591.107,A -85,B 0,C 180,E1 -20232.972,E2 -20232.972} C_VEL
LIN {X 0,Y 220.551,Z 599.15,A -85,B 0,C 180,E1 -20235.703,E2 -20235.703} C_VEL
LIN {X 0,Y 219.67,Z 604.578,A -85,B 0,C 180,E1 -20237.998,E2 -20237.998} C_VEL
LIN {X 0,Y 219.05,Z 609.882,A -85,B 0,C 180,E1 -20240.769,E2 -20240.769} C_VEL
LIN {X 0,Y 218.77,Z 613.98,A -85,B 0,C 180,E1 -20243.544,E2 -20243.544} C_VEL
LIN {X 0,Y 218.691,Z 616.987,A -85,B 0,C 180,E1 -20246.315,E2 -20246.315} C_VEL
LIN {X 0,Y 218.798,Z 618.444,A -85,B 0,C 180,E1 -20248.159,E2 -20248.159} C_VEL
LIN {X 0,Y 218.811,Z 619.45,A -85,B 0,C 180,E1 -20250,E2 -20250} C_VEL
LIN {X 0,Y 218.762,Z 620.053,A -85,B 0,C 180,E1 -20251.841,E2 -20251.841} C_VEL
LIN {X 0,Y 218.638,Z 620.171,A -85,B 0,C 180,E1 -20254.81,E2 -20254.81} C_VEL
LIN {X 0,Y 218.747,Z 619.453,A -85,B 0,C 180,E1 -20257.384,E2 -20257.384} C_VEL
LIN {X 0,Y 219.537,Z 617.082,A -85,B 0,C 180,E1 -20261.074,E2 -20261.074} C_VEL
LIN {X 0,Y 220.576,Z 614.21,A -85,B 0,C 180,E1 -20263.825,E2 -20263.825} C_VEL
LIN {X 0,Y 222.307,Z 610.347,A -85,B 0,C 180,E1 -20266.53,E2 -20266.53} C_VEL
LIN {X 0,Y 224.428,Z 605.388,A -85,B 0,C 180,E1 -20269.196,E2 -20269.196} C_VEL
LIN {X 0,Y 227.478,Z 598.029,A -85,B 0,C 180,E1 -20272.238,E2 -20272.238} C_VEL
LIN {X 0,Y 230.589,Z 590.042,A -85,B 0,C 180,E1 -20274.776,E2 -20274.776} C_VEL
LIN {X 0,Y 234.356,Z 580.149,A -85,B 0,C 180,E1 -20277.214,E2 -20277.214} C_VEL
LIN {X 0,Y 237.882,Z 569.802,A -85,B 0,C 180,E1 -20279.174,E2 -20279.174} C_VEL
LIN {X 0,Y 240.932,Z 559.602,A -85,B 0,C 180,E1 -20280.695,E2 -20280.695} C_VEL
LIN {X 0,Y 243.771,Z 548.49,A -85,B 0,C 180,E1 -20281.988,E2 -20281.988} C_VEL
LIN {X 0,Y 246.343,Z 536.1,A -85,B 0,C 180,E1 -20283.066,E2 -20283.066} C_VEL
LIN {X 0,Y 248.148,Z 523.885,A -85,B 0,C 180,E1 -20283.827,E2 -20283.827} C_VEL
LIN {X 0,Y 249.454,Z 510.008,A -85,B 0,C 180,E1 -20284.374,E2 -20284.374} C_VEL
LIN {X 0,Y 251.44,Z 468.334,A -85,B 0,C 180,E1 -20285.561,E2 -20285.561} C_VEL
LIN {X 0,Y 249.197,Z 451.614,A -85,B 0,C 180,E1 -20286.66,E2 -20286.66} C_VEL
LIN {X 0,Y 243.246,Z 438.502,A -85,B 0,C 180,E1 -20288.482,E2 -20288.482} C_VEL
LIN {X 0,Y 236.812,Z 425.924,A -85,B 0,C 180,E1 -20290.57,E2 -20290.57} C_VEL
LIN {X 0,Y 232.928,Z 419.2,A -85,B 0,C 180,E1 -20291.889,E2 -20291.889} C_VEL
LIN {X 0,Y 230.531,Z 415.153,A -85,B 0,C 180,E1 -20292.744,E2 -20292.744} C_VEL
LIN {X 0,Y 227.345,Z 410.064,A -85,B 0,C 180,E1 -20293.919,E2 -20293.919} C_VEL
LIN {X 0,Y 224.426,Z 405.517,A -85,B 0,C 180,E1 -20295.045,E2 -20295.045} C_VEL
LIN {X 0,Y 224.073,Z 404.686,A -85,B 0,C 180,E1 -20295.272,E2 -20295.272} C_VEL
LIN {X 0,Y 222.195,Z 398.437,A -85,B 0,C 180,E1 -20299.385,E2 -20299.385} C_VEL
LIN {X 0,Y 220.853,Z 393.968,A -85,B 0,C 180,E1 -20302.799,E2 -20302.799} C_VEL
LIN {X 0,Y 220.821,Z 393.971,A -85,B 0,C 180,E1 -20307.245,E2 -20307.245} C_VEL
LIN {X 0,Y 220.834,Z 393.973,A -85,B 0,C 180,E1 -20311.486,E2 -20311.486} C_VEL
LIN {X 0,Y 220.863,Z 393.97,A -85,B 0,C 180,E1 -20315.565,E2 -20315.565} C_VEL
LIN {X 0,Y 220.888,Z 393.963,A -85,B 0,C 180,E1 -20319.514,E2 -20319.514} C_VEL
LIN {X 0,Y 221.01,Z 393.942,A -85,B 0,C 180,E1 -20323.37,E2 -20323.37} C_VEL
LIN {X 0,Y 221.102,Z 393.937,A -85,B 0,C 180,E1 -20329.006,E2 -20329.006} C_VEL
LIN {X 0,Y 221.283,Z 393.904,A -85,B 0,C 180,E1 -20332.702,E2 -20332.702} C_VEL
LIN {X 0,Y 221.508,Z 393.879,A -85,B 0,C 180,E1 -20338.182,E2 -20338.182} C_VEL
LIN {X 0,Y 221.508,Z 393.879,A -85,B 0,C 180,E1 -20341.819,E2 -20341.819} C_VEL
LIN {X 0,Y 221.255,Z 393.91,A -85,B 0,C 180,E1 -20347.3,E2 -20347.3} C_VEL
LIN {X 0,Y 221.063,Z 393.939,A -85,B 0,C 180,E1 -20350.997,E2 -20350.997} C_VEL
LIN {X 0,Y 221.021,Z 393.942,A -85,B 0,C 180,E1 -20356.63,E2 -20356.63} C_VEL
LIN {X 0,Y 220.917,Z 393.956,A -85,B 0,C 180,E1 -20360.484,E2 -20360.484} C_VEL
LIN {X 0,Y 220.872,Z 393.964,A -85,B 0,C 180,E1 -20364.435,E2 -20364.435} C_VEL
LIN {X 0,Y 220.871,Z 394.134,A -85,B 0,C 180,E1 -20367.876,E2 -20367.876} C_VEL
LIN {X 0,Y 221.695,Z 396.607,A -85,B 0,C 180,E1 -20368.289,E2 -20368.289} C_VEL
LIN {X 0,Y 223.849,Z 398.932,A -85,B 0,C 180,E1 -20369.121,E2 -20369.121} C_VEL
LIN {X 0,Y 224.599,Z 399.667,A -85,B 0,C 180,E1 -20369.399,E2 -20369.399} C_VEL
LIN {X 0,Y 226.587,Z 402.835,A -85,B 0,C 180,E1 -20370.182,E2 -20370.182} C_VEL
LIN {X 0,Y 228.191,Z 404.616,A -85,B 0,C 180,E1 -20370.756,E2 -20370.756} C_VEL
LIN {X 0,Y 230.919,Z 408.357,A -85,B 0,C 180,E1 -20371.733,E2 -20371.733} C_VEL
LIN {X 0,Y 237.334,Z 417.67,A -85,B 0,C 180,E1 -20373.886,E2 -20373.886} C_VEL
LIN {X 0,Y 243.124,Z 426.833,A -85,B 0,C 180,E1 -20375.694,E2 -20375.694} C_VEL
LIN {X 0,Y 249.533,Z 439.295,A -85,B 0,C 180,E1 -20377.618,E2 -20377.618} C_VEL
LIN {X 0,Y 252.539,Z 445.893,A -85,B 0,C 180,E1 -20378.494,E2 -20378.494} C_VEL
LIN {X 0,Y 249.871,Z 497.264,A -85,B 0,C 180,E1 -20379.963,E2 -20379.963} C_VEL
LIN {X 0,Y 248.459,Z 510.734,A -85,B 0,C 180,E1 -20380.648,E2 -20380.648} C_VEL
LIN {X 0,Y 246.514,Z 523.405,A -85,B 0,C 180,E1 -20381.61,E2 -20381.61} C_VEL
LIN {X 0,Y 244.207,Z 534.742,A -85,B 0,C 180,E1 -20382.791,E2 -20382.791} C_VEL
LIN {X 0,Y 241.392,Z 546.042,A -85,B 0,C 180,E1 -20384.328,E2 -20384.328} C_VEL
LIN {X 0,Y 238.268,Z 556.441,A -85,B 0,C 180,E1 -20386.12,E2 -20386.12} C_VEL
LIN {X 0,Y 234.868,Z 566.351,A -85,B 0,C 180,E1 -20388.316,E2 -20388.316} C_VEL
LIN {X 0,Y 231.866,Z 574.08,A -85,B 0,C 180,E1 -20390.468,E2 -20390.468} C_VEL
LIN {X 0,Y 228.838,Z 581.27,A -85,B 0,C 180,E1 -20392.989,E2 -20392.989} C_VEL
LIN {X 0,Y 225.906,Z 587.782,A -85,B 0,C 180,E1 -20395.946,E2 -20395.946} C_VEL
LIN {X 0,Y 223.607,Z 592.428,A -85,B 0,C 180,E1 -20398.763,E2 -20398.763} C_VEL
LIN {X 0,Y 221.813,Z 595.878,A -85,B 0,C 180,E1 -20401.624,E2 -20401.624} C_VEL
LIN {X 0,Y 220.818,Z 597.556,A -85,B 0,C 180,E1 -20403.54,E2 -20403.54} C_VEL
LIN {X 0,Y 220.019,Z 598.8,A -85,B 0,C 180,E1 -20405.465,E2 -20405.465} C_VEL
LIN {X 0,Y 219.154,Z 599.82,A -85,B 0,C 180,E1 -20408.436,E2 -20408.436} C_VEL
LIN {X 0,Y 218.626,Z 599.836,A -85,B 0,C 180,E1 -20411.249,E2 -20411.249} C_VEL
LIN {X 0,Y 218.472,Z 598.558,A -85,B 0,C 180,E1 -20414.814,E2 -20414.814} C_VEL
LIN {X 0,Y 218.55,Z 597.032,A -85,B 0,C 180,E1 -20416.991,E2 -20416.991} C_VEL
LIN {X 0,Y 218.907,Z 594.169,A -85,B 0,C 180,E1 -20419.83,E2 -20419.83} C_VEL
LIN {X 0,Y 219.601,Z 590.004,A -85,B 0,C 180,E1 -20422.803,E2 -20422.803} C_VEL
LIN {X 0,Y 220.397,Z 585.201,A -85,B 0,C 180,E1 -20425.428,E2 -20425.428} C_VEL
LIN {X 0,Y 221.504,Z 578.862,A -85,B 0,C 180,E1 -20428.182,E2 -20428.182} C_VEL
LIN {X 0,Y 223.084,Z 570.893,A -85,B 0,C 180,E1 -20430.903,E2 -20430.903} C_VEL
LIN {X 0,Y 224.612,Z 562.781,A -85,B 0,C 180,E1 -20433.139,E2 -20433.139} C_VEL
LIN {X 0,Y 226.544,Z 552.847,A -85,B 0,C 180,E1 -20435.34,E2 -20435.34} C_VEL
LIN {X 0,Y 228.3,Z 541.762,A -85,B 0,C 180,E1 -20437.295,E2 -20437.295} C_VEL
LIN {X 0,Y 229.927,Z 530.852,A -85,B 0,C 180,E1 -20438.791,E2 -20438.791} C_VEL
LIN {X 0,Y 231.361,Z 518.848,A -85,B 0,C 180,E1 -20440.059,E2 -20440.059} C_VEL
LIN {X 0,Y 232.494,Z 505.765,A -85,B 0,C 180,E1 -20441.055,E2 -20441.055} C_VEL
LIN {X 0,Y 233.188,Z 492.802,A -85,B 0,C 180,E1 -20441.683,E2 -20441.683} C_VEL
LIN {X 0,Y 235.592,Z 429.468,A -85,B 0,C 180,E1 -20443.555,E2 -20443.555} C_VEL
LIN {X 0,Y 233.146,Z 421.57,A -85,B 0,C 180,E1 -20444.093,E2 -20444.093} C_VEL
LIN {X 0,Y 228.589,Z 410.41,A -85,B 0,C 180,E1 -20445.009,E2 -20445.009} C_VEL
LIN {X 0,Y 221.833,Z 396.48,A -85,B 0,C 180,E1 -20446.354,E2 -20446.354} C_VEL
LIN {X 0,Y 221.005,Z 393.958,A -85,B 0,C 180,E1 -20446.586,E2 -20446.586} C_VEL
LIN {X 0,Y 220.896,Z 393.969,A -85,B 0,C 180,E1 -20450.485,E2 -20450.485} C_VEL
LIN {X 0,Y 220.87,Z 393.961,A -85,B 0,C 180,E1 -20454.434,E2 -20454.434} C_VEL
LIN {X 0,Y 220.839,Z 393.976,A -85,B 0,C 180,E1 -20458.512,E2 -20458.512} C_VEL
LIN {X 0,Y 220.819,Z 393.976,A -85,B 0,C 180,E1 -20462.755,E2 -20462.755} C_VEL
LIN {X 0,Y 220.811,Z 393.977,A -85,B 0,C 180,E1 -20467.277,E2 -20467.277} C_VEL
LIN {X 0,Y 220.771,Z 393.978,A -85,B 0,C 180,E1 -20471.951,E2 -20471.951} C_VEL
LIN {X 0,Y 220.775,Z 393.979,A -85,B 0,C 180,E1 -20475.545,E2 -20475.545} C_VEL
LIN {X 0,Y 220.806,Z 393.979,A -85,B 0,C 180,E1 -20480.462,E2 -20480.462} C_VEL
LIN {X 0,Y 220.799,Z 393.981,A -85,B 0,C 180,E1 -20485.044,E2 -20485.044} C_VEL
LIN {X 0,Y 220.866,Z 393.966,A -85,B 0,C 180,E1 -20489.394,E2 -20489.394} C_VEL
LIN {X 0,Y 220.893,Z 393.968,A -85,B 0,C 180,E1 -20493.549,E2 -20493.549} C_VEL
LIN {X 0,Y 220.875,Z 393.967,A -85,B 0,C 180,E1 -20497.552,E2 -20497.552} C_VEL
LIN {X 0,Y 220.981,Z 393.952,A -85,B 0,C 180,E1 -20502.571,E2 -20502.571} C_VEL
LIN {X 0,Y 221.007,Z 393.953,A -85,B 0,C 180,E1 -20507.138,E2 -20507.138} C_VEL
LIN {X 0,Y 221.2,Z 393.923,A -85,B 0,C 180,E1 -20510.859,E2 -20510.859} C_VEL
LIN {X 0,Y 221.267,Z 393.92,A -85,B 0,C 180,E1 -20512.7,E2 -20512.7} C_VEL
LIN {X 0,Y 221.508,Z 393.881,A -85,B 0,C 180,E1 -20518.181,E2 -20518.181} C_VEL
LIN {X 0,Y 221.507,Z 393.86,A -85,B 0,C 180,E1 -20521.818,E2 -20521.818} C_VEL
LIN {X 0,Y 221.254,Z 393.922,A -85,B 0,C 180,E1 -20527.299,E2 -20527.299} C_VEL
LIN {X 0,Y 221.062,Z 393.941,A -85,B 0,C 180,E1 -20530.996,E2 -20530.996} C_VEL
LIN {X 0,Y 221.011,Z 393.952,A -85,B 0,C 180,E1 -20536.63,E2 -20536.63} C_VEL
LIN {X 0,Y 220.888,Z 393.971,A -85,B 0,C 180,E1 -20540.486,E2 -20540.486} C_VEL
LIN {X 0,Y 220.863,Z 393.973,A -85,B 0,C 180,E1 -20544.435,E2 -20544.435} C_VEL
LIN {X 0,Y 220.834,Z 393.977,A -85,B 0,C 180,E1 -20548.514,E2 -20548.514} C_VEL
LIN {X 0,Y 220.821,Z 393.98,A -85,B 0,C 180,E1 -20552.755,E2 -20552.755} C_VEL
LIN {X 0,Y 220.835,Z 393.98,A -85,B 0,C 180,E1 -20557.288,E2 -20557.288} C_VEL
LIN {X 0,Y 220.848,Z 393.981,A -85,B 0,C 180,E1 -20560.154,E2 -20560.154} C_VEL
LIN {X 0,Y 220.186,Z 394.067,A -85,B 0,C 180,E1 -20561.674,E2 -20561.674} C_VEL
LIN {X 0,Y 217.292,Z 394.423,A -85,B 0,C 180,E1 -20564.153,E2 -20564.153} C_VEL
LIN {X 0,Y 214.841,Z 394.727,A -85,B 0,C 180,E1 -20566.178,E2 -20566.178} C_VEL
LIN {X 0,Y 213.819,Z 394.853,A -85,B 0,C 180,E1 -20567.753,E2 -20567.753} C_VEL
LIN {X 0,Y 213.753,Z 394.854,A -85,B 0,C 180,E1 -20568.286,E2 -20568.286} C_VEL
LIN {X 0,Y 213.849,Z 394.872,A -85,B 0,C 180,E1 -20571.21,E2 -20571.21} C_VEL
LIN {X 0,Y 215.883,Z 403.956,A -85,B 0,C 180,E1 -20575.318,E2 -20575.318} C_VEL
LIN {X 0,Y 216.465,Z 407.078,A -85,B 0,C 180,E1 -20576.656,E2 -20576.656} C_VEL
LIN {X 0,Y 223.906,Z 426.815,A -85,B 0,C 180,E1 -20578.338,E2 -20578.338} C_VEL
LIN {X 0,Y 228.018,Z 464.639,A -85,B 0,C 180,E1 -20580.139,E2 -20580.139} C_VEL
LIN {X 0,Y 226.122,Z 515.84,A -85,B 0,C 180,E1 -20581.734,E2 -20581.734} C_VEL
LIN {X 0,Y 225.105,Z 529.623,A -85,B 0,C 180,E1 -20582.518,E2 -20582.518} C_VEL
LIN {X 0,Y 223.682,Z 541.705,A -85,B 0,C 180,E1 -20583.528,E2 -20583.528} C_VEL
LIN {X 0,Y 221.904,Z 553.925,A -85,B 0,C 180,E1 -20584.938,E2 -20584.938} C_VEL
LIN {X 0,Y 219.78,Z 565.516,A -85,B 0,C 180,E1 -20586.69,E2 -20586.69} C_VEL
LIN {X 0,Y 217.896,Z 575.999,A -85,B 0,C 180,E1 -20588.725,E2 -20588.725} C_VEL
LIN {X 0,Y 215.975,Z 585.366,A -85,B 0,C 180,E1 -20591.01,E2 -20591.01} C_VEL
LIN {X 0,Y 214.843,Z 591.682,A -85,B 0,C 180,E1 -20592.878,E2 -20592.878} C_VEL
LIN {X 0,Y 213.391,Z 599.512,A -85,B 0,C 180,E1 -20595.7,E2 -20595.7} C_VEL
LIN {X 0,Y 212.4,Z 605.775,A -85,B 0,C 180,E1 -20598.549,E2 -20598.549} C_VEL
LIN {X 0,Y 211.872,Z 610.737,A -85,B 0,C 180,E1 -20601.416,E2 -20601.416} C_VEL
LIN {X 0,Y 211.635,Z 614.533,A -85,B 0,C 180,E1 -20604.283,E2 -20604.283} C_VEL
LIN {X 0,Y 211.596,Z 616.478,A -85,B 0,C 180,E1 -20606.191,E2 -20606.191} C_VEL
LIN {X 0,Y 211.704,Z 617.994,A -85,B 0,C 180,E1 -20608.098,E2 -20608.098} C_VEL
LIN {X 0,Y 211.743,Z 619.038,A -85,B 0,C 180,E1 -20610,E2 -20610} C_VEL
LIN {X 0,Y 211.668,Z 619.671,A -85,B 0,C 180,E1 -20611.903,E2 -20611.903} C_VEL
LIN {X 0,Y 211.568,Z 619.764,A -85,B 0,C 180,E1 -20615.719,E2 -20615.719} C_VEL
LIN {X 0,Y 212.018,Z 618.235,A -85,B 0,C 180,E1 -20619.54,E2 -20619.54} C_VEL
LIN {X 0,Y 213.206,Z 615.146,A -85,B 0,C 180,E1 -20623.341,E2 -20623.341} C_VEL
LIN {X 0,Y 214.842,Z 611.687,A -85,B 0,C 180,E1 -20626.144,E2 -20626.144} C_VEL
LIN {X 0,Y 216.913,Z 607.181,A -85,B 0,C 180,E1 -20628.905,E2 -20628.905} C_VEL
LIN {X 0,Y 219.467,Z 601.55,A -85,B 0,C 180,E1 -20631.587,E2 -20631.587} C_VEL
LIN {X 0,Y 222.472,Z 594.449,A -85,B 0,C 180,E1 -20634.247,E2 -20634.247} C_VEL
LIN {X 0,Y 226.084,Z 585.682,A -85,B 0,C 180,E1 -20636.791,E2 -20636.791} C_VEL
LIN {X 0,Y 229.873,Z 575.761,A -85,B 0,C 180,E1 -20639.035,E2 -20639.035} C_VEL
LIN {X 0,Y 233.283,Z 565.692,A -85,B 0,C 180,E1 -20640.806,E2 -20640.806} C_VEL
LIN {X 0,Y 236.54,Z 554.553,A -85,B 0,C 180,E1 -20642.33,E2 -20642.33} C_VEL
LIN {X 0,Y 239.588,Z 542.078,A -85,B 0,C 180,E1 -20643.619,E2 -20643.619} C_VEL
LIN {X 0,Y 241.863,Z 529.357,A -85,B 0,C 180,E1 -20644.578,E2 -20644.578} C_VEL
LIN {X 0,Y 243.465,Z 517,A -85,B 0,C 180,E1 -20645.199,E2 -20645.199} C_VEL
LIN {X 0,Y 244.785,Z 495.645,A -85,B 0,C 180,E1 -20645.859,E2 -20645.859} C_VEL
LIN {X 0,Y 246.163,Z 470.06,A -85,B 0,C 180,E1 -20646.575,E2 -20646.575} C_VEL
LIN {X 0,Y 244.232,Z 455.04,A -85,B 0,C 180,E1 -20647.589,E2 -20647.589} C_VEL
LIN {X 0,Y 239.013,Z 443.069,A -85,B 0,C 180,E1 -20649.285,E2 -20649.285} C_VEL
LIN {X 0,Y 232.542,Z 430.228,A -85,B 0,C 180,E1 -20651.491,E2 -20651.491} C_VEL
LIN {X 0,Y 226.945,Z 420.425,A -85,B 0,C 180,E1 -20653.529,E2 -20653.529} C_VEL
LIN {X 0,Y 223.452,Z 414.885,A -85,B 0,C 180,E1 -20654.875,E2 -20654.875} C_VEL
LIN {X 0,Y 220.094,Z 409.597,A -85,B 0,C 180,E1 -20656.247,E2 -20656.247} C_VEL
LIN {X 0,Y 217.161,Z 405.215,A -85,B 0,C 180,E1 -20657.509,E2 -20657.509} C_VEL
LIN {X 0,Y 216.682,Z 404.109,A -85,B 0,C 180,E1 -20657.807,E2 -20657.807} C_VEL
LIN {X 0,Y 214.994,Z 398.829,A -85,B 0,C 180,E1 -20661.677,E2 -20661.677} C_VEL
LIN {X 0,Y 213.765,Z 394.856,A -85,B 0,C 180,E1 -20665.011,E2 -20665.011} C_VEL
LIN {X 0,Y 213.793,Z 394.849,A -85,B 0,C 180,E1 -20668.724,E2 -20668.724} C_VEL
LIN {X 0,Y 213.822,Z 394.845,A -85,B 0,C 180,E1 -20672.603,E2 -20672.603} C_VEL
LIN {X 0,Y 213.848,Z 394.84,A -85,B 0,C 180,E1 -20676.953,E2 -20676.953} C_VEL
LIN {X 0,Y 213.928,Z 394.823,A -85,B 0,C 180,E1 -20682.306,E2 -20682.306} C_VEL
LIN {X 0,Y 213.947,Z 394.823,A -85,B 0,C 180,E1 -20686.707,E2 -20686.707} C_VEL
LIN {X 0,Y 214.163,Z 394.807,A -85,B 0,C 180,E1 -20690.557,E2 -20690.557} C_VEL
LIN {X 0,Y 214.222,Z 394.784,A -85,B 0,C 180,E1 -20692.46,E2 -20692.46} C_VEL
LIN {X 0,Y 214.441,Z 394.758,A -85,B 0,C 180,E1 -20698.122,E2 -20698.122} C_VEL
LIN {X 0,Y 214.55,Z 394.761,A -85,B 0,C 180,E1 -20700,E2 -20700} C_VEL
LIN {X 0,Y 214.441,Z 394.759,A -85,B 0,C 180,E1 -20701.879,E2 -20701.879} C_VEL
LIN {X 0,Y 214.194,Z 394.789,A -85,B 0,C 180,E1 -20707.542,E2 -20707.542} C_VEL
LIN {X 0,Y 213.995,Z 394.816,A -85,B 0,C 180,E1 -20711.365,E2 -20711.365} C_VEL
LIN {X 0,Y 213.932,Z 394.829,A -85,B 0,C 180,E1 -20715.238,E2 -20715.238} C_VEL
LIN {X 0,Y 213.879,Z 394.838,A -85,B 0,C 180,E1 -20719.184,E2 -20719.184} C_VEL
LIN {X 0,Y 213.857,Z 394.839,A -85,B 0,C 180,E1 -20723.227,E2 -20723.227} C_VEL
LIN {X 0,Y 213.811,Z 394.849,A -85,B 0,C 180,E1 -20725.298,E2 -20725.298} C_VEL
LIN {X 0,Y 214.631,Z 397.359,A -85,B 0,C 180,E1 -20725.779,E2 -20725.779} C_VEL
LIN {X 0,Y 216.667,Z 399.674,A -85,B 0,C 180,E1 -20726.681,E2 -20726.681} C_VEL
LIN {X 0,Y 217.636,Z 400.35,A -85,B 0,C 180,E1 -20727.073,E2 -20727.073} C_VEL
LIN {X 0,Y 219.515,Z 403.595,A -85,B 0,C 180,E1 -20727.92,E2 -20727.92} C_VEL
LIN {X 0,Y 221.574,Z 405.808,A -85,B 0,C 180,E1 -20728.734,E2 -20728.734} C_VEL
LIN {X 0,Y 224.222,Z 409.419,A -85,B 0,C 180,E1 -20729.776,E2 -20729.776} C_VEL
LIN {X 0,Y 231.212,Z 419.267,A -85,B 0,C 180,E1 -20732.33,E2 -20732.33} C_VEL
LIN {X 0,Y 238.148,Z 430.083,A -85,B 0,C 180,E1 -20734.633,E2 -20734.633} C_VEL
LIN {X 0,Y 244.217,Z 441.806,A -85,B 0,C 180,E1 -20736.562,E2 -20736.562} C_VEL
LIN {X 0,Y 247.209,Z 448.5,A -85,B 0,C 180,E1 -20737.485,E2 -20737.485} C_VEL
LIN {X 0,Y 244.474,Z 497.687,A -85,B 0,C 180,E1 -20738.902,E2 -20738.902} C_VEL
LIN {X 0,Y 243.043,Z 510.905,A -85,B 0,C 180,E1 -20739.582,E2 -20739.582} C_VEL
LIN {X 0,Y 241.143,Z 522.925,A -85,B 0,C 180,E1 -20740.497,E2 -20740.497} C_VEL
LIN {X 0,Y 238.774,Z 534.39,A -85,B 0,C 180,E1 -20741.681,E2 -20741.681} C_VEL
LIN {X 0,Y 236.055,Z 545.015,A -85,B 0,C 180,E1 -20743.113,E2 -20743.113} C_VEL
LIN {X 0,Y 232.889,Z 555.182,A -85,B 0,C 180,E1 -20744.834,E2 -20744.834} C_VEL
LIN {X 0,Y 229.352,Z 565.27,A -85,B 0,C 180,E1 -20747.017,E2 -20747.017} C_VEL
LIN {X 0,Y 226.104,Z 573.401,A -85,B 0,C 180,E1 -20749.252,E2 -20749.252} C_VEL
LIN {X 0,Y 222.979,Z 580.547,A -85,B 0,C 180,E1 -20751.736,E2 -20751.736} C_VEL
LIN {X 0,Y 219.705,Z 587.45,A -85,B 0,C 180,E1 -20754.846,E2 -20754.846} C_VEL
LIN {X 0,Y 217.084,Z 592.487,A -85,B 0,C 180,E1 -20757.876,E2 -20757.876} C_VEL
LIN {X 0,Y 215.23,Z 595.874,A -85,B 0,C 180,E1 -20760.673,E2 -20760.673} C_VEL
LIN {X 0,Y 214.144,Z 597.627,A -85,B 0,C 180,E1 -20762.648,E2 -20762.648} C_VEL
LIN {X 0,Y 213.217,Z 598.933,A -85,B 0,C 180,E1 -20764.628,E2 -20764.628} C_VEL
LIN {X 0,Y 212.157,Z 600.157,A -85,B 0,C 180,E1 -20768.057,E2 -20768.057} C_VEL
LIN {X 0,Y 211.619,Z 600.211,A -85,B 0,C 180,E1 -20770.604,E2 -20770.604} C_VEL
LIN {X 0,Y 211.405,Z 599.794,A -85,B 0,C 180,E1 -20772.591,E2 -20772.591} C_VEL
LIN {X 0,Y 211.393,Z 598.918,A -85,B 0,C 180,E1 -20774.613,E2 -20774.613} C_VEL
LIN {X 0,Y 211.416,Z 597.645,A -85,B 0,C 180,E1 -20776.544,E2 -20776.544} C_VEL
LIN {X 0,Y 211.762,Z 594.901,A -85,B 0,C 180,E1 -20779.483,E2 -20779.483} C_VEL
LIN {X 0,Y 212.505,Z 590.456,A -85,B 0,C 180,E1 -20782.83,E2 -20782.83} C_VEL
LIN {X 0,Y 213.214,Z 586.202,A -85,B 0,C 180,E1 -20785.273,E2 -20785.273} C_VEL
LIN {X 0,Y 214.351,Z 580.012,A -85,B 0,C 180,E1 -20788.121,E2 -20788.121} C_VEL
LIN {X 0,Y 215.917,Z 572.305,A -85,B 0,C 180,E1 -20790.932,E2 -20790.932} C_VEL
LIN {X 0,Y 217.518,Z 564.402,A -85,B 0,C 180,E1 -20793.241,E2 -20793.241} C_VEL
LIN {X 0,Y 219.423,Z 554.74,A -85,B 0,C 180,E1 -20795.514,E2 -20795.514} C_VEL
LIN {X 0,Y 221.243,Z 544.051,A -85,B 0,C 180,E1 -20797.529,E2 -20797.529} C_VEL
LIN {X 0,Y 222.897,Z 533.685,A -85,B 0,C 180,E1 -20799.07,E2 -20799.07} C_VEL
LIN {X 0,Y 224.491,Z 521.317,A -85,B 0,C 180,E1 -20800.484,E2 -20800.484} C_VEL
LIN {X 0,Y 225.704,Z 508.353,A -85,B 0,C 180,E1 -20801.563,E2 -20801.563} C_VEL
LIN {X 0,Y 226.514,Z 495.749,A -85,B 0,C 180,E1 -20802.259,E2 -20802.259} C_VEL
LIN {X 0,Y 229.034,Z 430.13,A -85,B 0,C 180,E1 -20804.273,E2 -20804.273} C_VEL
LIN {X 0,Y 224.397,Z 417.328,A -85,B 0,C 180,E1 -20805.279,E2 -20805.279} C_VEL
LIN {X 0,Y 216.457,Z 400.527,A -85,B 0,C 180,E1 -20806.923,E2 -20806.923} C_VEL
LIN {X 0,Y 214.131,Z 395.782,A -85,B 0,C 180,E1 -20807.424,E2 -20807.424} C_VEL
LIN {X 0,Y 213.94,Z 394.838,A -85,B 0,C 180,E1 -20807.535,E2 -20807.535} C_VEL
LIN {X 0,Y 213.85,Z 394.838,A -85,B 0,C 180,E1 -20813.226,E2 -20813.226} C_VEL
LIN {X 0,Y 213.831,Z 394.851,A -85,B 0,C 180,E1 -20817.449,E2 -20817.449} C_VEL
LIN {X 0,Y 213.779,Z 394.854,A -85,B 0,C 180,E1 -20821.735,E2 -20821.735} C_VEL
LIN {X 0,Y 213.745,Z 394.857,A -85,B 0,C 180,E1 -20826.287,E2 -20826.287} C_VEL
LIN {X 0,Y 213.713,Z 394.858,A -85,B 0,C 180,E1 -20831.124,E2 -20831.124} C_VEL
LIN {X 0,Y 213.707,Z 394.862,A -85,B 0,C 180,E1 -20833.677,E2 -20833.677} C_VEL
LIN {X 0,Y 213.707,Z 394.859,A -85,B 0,C 180,E1 -20836.342,E2 -20836.342} C_VEL
LIN {X 0,Y 213.717,Z 394.863,A -85,B 0,C 180,E1 -20839.142,E2 -20839.142} C_VEL
LIN {X 0,Y 213.742,Z 394.855,A -85,B 0,C 180,E1 -20843.711,E2 -20843.711} C_VEL
LIN {X 0,Y 213.779,Z 394.85,A -85,B 0,C 180,E1 -20848.73,E2 -20848.73} C_VEL
LIN {X 0,Y 213.824,Z 394.85,A -85,B 0,C 180,E1 -20852.602,E2 -20852.602} C_VEL
LIN {X 0,Y 213.849,Z 394.84,A -85,B 0,C 180,E1 -20856.952,E2 -20856.952} C_VEL
LIN {X 0,Y 213.94,Z 394.827,A -85,B 0,C 180,E1 -20862.803,E2 -20862.803} C_VEL
LIN {X 0,Y 213.949,Z 394.834,A -85,B 0,C 180,E1 -20866.706,E2 -20866.706} C_VEL
LIN {X 0,Y 214.138,Z 394.803,A -85,B 0,C 180,E1 -20870.555,E2 -20870.555} C_VEL
LIN {X 0,Y 214.204,Z 394.797,A -85,B 0,C 180,E1 -20872.458,E2 -20872.458} C_VEL
LIN {X 0,Y 214.441,Z 394.761,A -85,B 0,C 180,E1 -20878.121,E2 -20878.121} C_VEL
LIN {X 0,Y 214.545,Z 394.733,A -85,B 0,C 180,E1 -20880,E2 -20880} C_VEL
LIN {X 0,Y 214.44,Z 394.738,A -85,B 0,C 180,E1 -20881.878,E2 -20881.878} C_VEL
LIN {X 0,Y 214.193,Z 394.802,A -85,B 0,C 180,E1 -20887.541,E2 -20887.541} C_VEL
LIN {X 0,Y 213.994,Z 394.821,A -85,B 0,C 180,E1 -20891.364,E2 -20891.364} C_VEL
LIN {X 0,Y 213.927,Z 394.836,A -85,B 0,C 180,E1 -20895.237,E2 -20895.237} C_VEL
LIN {X 0,Y 213.835,Z 394.845,A -85,B 0,C 180,E1 -20899.187,E2 -20899.187} C_VEL
LIN {X 0,Y 213.843,Z 394.843,A -85,B 0,C 180,E1 -20903.227,E2 -20903.227} C_VEL
LIN {X 0,Y 213.825,Z 394.848,A -85,B 0,C 180,E1 -20907.45,E2 -20907.45} C_VEL
LIN {X 0,Y 213.776,Z 394.857,A -85,B 0,C 180,E1 -20911.736,E2 -20911.736} C_VEL
LIN {X 0,Y 213.751,Z 394.862,A -85,B 0,C 180,E1 -20916.287,E2 -20916.287} C_VEL
LIN {X 0,Y 213.791,Z 394.858,A -85,B 0,C 180,E1 -20921.106,E2 -20921.106} C_VEL
LIN {X 0,Y 213.806,Z 394.857,A -85,B 0,C 180,E1 -20923.685,E2 -20923.685} C_VEL
LIN {X 0,Y 213.809,Z 394.854,A -85,B 0,C 180,E1 -20926.349,E2 -20926.349} C_VEL
LIN {X 0,Y 213.753,Z 394.854,A -85,B 0,C 180,E1 -20928.286,E2 -20928.286} C_VEL
LIN {X 0,Y 213.178,Z 395.236,A -85,B 0,C 180,E1 -20929.34,E2 -20929.34} C_VEL
LIN {X 0,Y 211.284,Z 396.647,A -85,B 0,C 180,E1 -20930.654,E2 -20930.654} C_VEL
LIN {X 0,Y 208.487,Z 400.05,A -85,B 0,C 180,E1 -20932.552,E2 -20932.552} C_VEL
LIN {X 0,Y 208.231,Z 402.092,A -85,B 0,C 180,E1 -20933.517,E2 -20933.517} C_VEL
LIN {X 0,Y 209.238,Z 406.784,A -85,B 0,C 180,E1 -20935.631,E2 -20935.631} C_VEL
LIN {X 0,Y 217.639,Z 428.799,A -85,B 0,C 180,E1 -20937.615,E2 -20937.615} C_VEL
LIN {X 0,Y 221.519,Z 464.317,A -85,B 0,C 180,E1 -20939.382,E2 -20939.382} C_VEL
LIN {X 0,Y 219.605,Z 515.56,A -85,B 0,C 180,E1 -20941.028,E2 -20941.028} C_VEL
LIN {X 0,Y 218.545,Z 529.139,A -85,B 0,C 180,E1 -20941.816,E2 -20941.816} C_VEL
LIN {X 0,Y 217.011,Z 541.832,A -85,B 0,C 180,E1 -20942.909,E2 -20942.909} C_VEL
LIN {X 0,Y 215.176,Z 553.917,A -85,B 0,C 180,E1 -20944.357,E2 -20944.357} C_VEL
LIN {X 0,Y 213.196,Z 564.134,A -85,B 0,C 180,E1 -20945.925,E2 -20945.925} C_VEL
LIN {X 0,Y 211.219,Z 574.8,A -85,B 0,C 180,E1 -20948.018,E2 -20948.018} C_VEL
LIN {X 0,Y 209.151,Z 584.362,A -85,B 0,C 180,E1 -20950.366,E2 -20950.366} C_VEL
LIN {X 0,Y 208.041,Z 590.752,A -85,B 0,C 180,E1 -20952.3,E2 -20952.3} C_VEL
LIN {X 0,Y 206.497,Z 598.729,A -85,B 0,C 180,E1 -20955.211,E2 -20955.211} C_VEL
LIN {X 0,Y 205.4,Z 605.076,A -85,B 0,C 180,E1 -20958.153,E2 -20958.153} C_VEL
LIN {X 0,Y 204.837,Z 610.117,A -85,B 0,C 180,E1 -20961.118,E2 -20961.118} C_VEL
LIN {X 0,Y 204.569,Z 613.987,A -85,B 0,C 180,E1 -20964.084,E2 -20964.084} C_VEL
LIN {X 0,Y 204.502,Z 615.964,A -85,B 0,C 180,E1 -20966.059,E2 -20966.059} C_VEL
LIN {X 0,Y 204.613,Z 617.522,A -85,B 0,C 180,E1 -20968.032,E2 -20968.032} C_VEL
LIN {X 0,Y 204.677,Z 618.625,A -85,B 0,C 180,E1 -20970,E2 -20970} C_VEL
LIN {X 0,Y 204.577,Z 619.288,A -85,B 0,C 180,E1 -20971.969,E2 -20971.969} C_VEL
LIN {X 0,Y 204.466,Z 619.585,A -85,B 0,C 180,E1 -20974.586,E2 -20974.586} C_VEL
LIN {X 0,Y 204.625,Z 618.937,A -85,B 0,C 180,E1 -20977.896,E2 -20977.896} C_VEL
LIN {X 0,Y 205.527,Z 616.695,A -85,B 0,C 180,E1 -20981.839,E2 -20981.839} C_VEL
LIN {X 0,Y 206.785,Z 613.96,A -85,B 0,C 180,E1 -20984.767,E2 -20984.767} C_VEL
LIN {X 0,Y 208.72,Z 610.242,A -85,B 0,C 180,E1 -20987.64,E2 -20987.64} C_VEL
LIN {X 0,Y 211.055,Z 605.442,A -85,B 0,C 180,E1 -20990.465,E2 -20990.465} C_VEL
LIN {X 0,Y 214.382,Z 598.303,A -85,B 0,C 180,E1 -20993.677,E2 -20993.677} C_VEL
LIN {X 0,Y 217.795,Z 590.58,A -85,B 0,C 180,E1 -20996.339,E2 -20996.339} C_VEL
LIN {X 0,Y 221.844,Z 580.94,A -85,B 0,C 180,E1 -20998.889,E2 -20998.889} C_VEL
LIN {X 0,Y 225.65,Z 571.02,A -85,B 0,C 180,E1 -21000.923,E2 -21000.923} C_VEL
LIN {X 0,Y 229.355,Z 559.86,A -85,B 0,C 180,E1 -21002.688,E2 -21002.688} C_VEL
LIN {X 0,Y 232.38,Z 548.974,A -85,B 0,C 180,E1 -21004.021,E2 -21004.021} C_VEL
LIN {X 0,Y 235.123,Z 536.966,A -85,B 0,C 180,E1 -21005.126,E2 -21005.126} C_VEL
LIN {X 0,Y 237.208,Z 524.678,A -85,B 0,C 180,E1 -21005.944,E2 -21005.944} C_VEL
LIN {X 0,Y 238.584,Z 512.2,A -85,B 0,C 180,E1 -21006.485,E2 -21006.485} C_VEL
LIN {X 0,Y 240.841,Z 470.452,A -85,B 0,C 180,E1 -21007.715,E2 -21007.715} C_VEL
LIN {X 0,Y 239.196,Z 457.758,A -85,B 0,C 180,E1 -21008.62,E2 -21008.62} C_VEL
LIN {X 0,Y 234.016,Z 445.982,A -85,B 0,C 180,E1 -21010.398,E2 -21010.398} C_VEL
LIN {X 0,Y 228.664,Z 435.183,A -85,B 0,C 180,E1 -21012.323,E2 -21012.323} C_VEL
LIN {X 0,Y 223.453,Z 425.759,A -85,B 0,C 180,E1 -21014.324,E2 -21014.324} C_VEL
LIN {X 0,Y 219.794,Z 419.863,A -85,B 0,C 180,E1 -21015.803,E2 -21015.803} C_VEL
LIN {X 0,Y 216.667,Z 414.905,A -85,B 0,C 180,E1 -21017.146,E2 -21017.146} C_VEL
LIN {X 0,Y 213.074,Z 409.309,A -85,B 0,C 180,E1 -21018.804,E2 -21018.804} C_VEL
LIN {X 0,Y 210.189,Z 405.397,A -85,B 0,C 180,E1 -21020.194,E2 -21020.194} C_VEL
LIN {X 0,Y 209.254,Z 403.546,A -85,B 0,C 180,E1 -21020.718,E2 -21020.718} C_VEL
LIN {X 0,Y 207.629,Z 398.551,A -85,B 0,C 180,E1 -21024.87,E2 -21024.87} C_VEL
LIN {X 0,Y 206.706,Z 395.731,A -85,B 0,C 180,E1 -21027.543,E2 -21027.543} C_VEL
LIN {X 0,Y 206.763,Z 395.729,A -85,B 0,C 180,E1 -21032.096,E2 -21032.096} C_VEL
LIN {X 0,Y 206.782,Z 395.724,A -85,B 0,C 180,E1 -21036.584,E2 -21036.584} C_VEL
LIN {X 0,Y 206.872,Z 395.703,A -85,B 0,C 180,E1 -21042.197,E2 -21042.197} C_VEL
LIN {X 0,Y 206.889,Z 395.706,A -85,B 0,C 180,E1 -21046.244,E2 -21046.244} C_VEL
LIN {X 0,Y 207.101,Z 395.688,A -85,B 0,C 180,E1 -21050.231,E2 -21050.231} C_VEL
LIN {X 0,Y 207.162,Z 395.663,A -85,B 0,C 180,E1 -21052.201,E2 -21052.201} C_VEL
LIN {X 0,Y 207.378,Z 395.638,A -85,B 0,C 180,E1 -21058.058,E2 -21058.058} C_VEL
LIN {X 0,Y 207.514,Z 395.637,A -85,B 0,C 180,E1 -21060,E2 -21060} C_VEL
LIN {X 0,Y 207.378,Z 395.638,A -85,B 0,C 180,E1 -21061.943,E2 -21061.943} C_VEL
LIN {X 0,Y 207.137,Z 395.669,A -85,B 0,C 180,E1 -21067.801,E2 -21067.801} C_VEL
LIN {X 0,Y 206.92,Z 395.696,A -85,B 0,C 180,E1 -21071.759,E2 -21071.759} C_VEL
LIN {X 0,Y 206.872,Z 395.705,A -85,B 0,C 180,E1 -21075.771,E2 -21075.771} C_VEL
LIN {X 0,Y 206.816,Z 395.713,A -85,B 0,C 180,E1 -21079.866,E2 -21079.866} C_VEL
LIN {X 0,Y 206.834,Z 395.857,A -85,B 0,C 180,E1 -21082.423,E2 -21082.423} C_VEL
LIN {X 0,Y 207.551,Z 398.102,A -85,B 0,C 180,E1 -21082.894,E2 -21082.894} C_VEL
LIN {X 0,Y 209.46,Z 400.451,A -85,B 0,C 180,E1 -21083.875,E2 -21083.875} C_VEL
LIN {X 0,Y 210.92,Z 401.471,A -85,B 0,C 180,E1 -21084.549,E2 -21084.549} C_VEL
LIN {X 0,Y 212.681,Z 404.496,A -85,B 0,C 180,E1 -21085.442,E2 -21085.442} C_VEL
LIN {X 0,Y 214.86,Z 406.804,A -85,B 0,C 180,E1 -21086.416,E2 -21086.416} C_VEL
LIN {X 0,Y 217.441,Z 410.409,A -85,B 0,C 180,E1 -21087.564,E2 -21087.564} C_VEL
LIN {X 0,Y 218.566,Z 411.786,A -85,B 0,C 180,E1 -21088.036,E2 -21088.036} C_VEL
LIN {X 0,Y 224.963,Z 420.701,A -85,B 0,C 180,E1 -21090.574,E2 -21090.574} C_VEL
LIN {X 0,Y 231.773,Z 430.967,A -85,B 0,C 180,E1 -21093.024,E2 -21093.024} C_VEL
LIN {X 0,Y 236.138,Z 438.651,A -85,B 0,C 180,E1 -21094.504,E2 -21094.504} C_VEL
LIN {X 0,Y 241.837,Z 450.624,A -85,B 0,C 180,E1 -21096.382,E2 -21096.382} C_VEL
LIN {X 0,Y 239.165,Z 498.043,A -85,B 0,C 180,E1 -21097.788,E2 -21097.788} C_VEL
LIN {X 0,Y 237.612,Z 511.823,A -85,B 0,C 180,E1 -21098.516,E2 -21098.516} C_VEL
LIN {X 0,Y 235.565,Z 524.036,A -85,B 0,C 180,E1 -21099.47,E2 -21099.47} C_VEL
LIN {X 0,Y 232.992,Z 535.706,A -85,B 0,C 180,E1 -21100.724,E2 -21100.724} C_VEL
LIN {X 0,Y 230.095,Z 546.4,A -85,B 0,C 180,E1 -21102.22,E2 -21102.22} C_VEL
LIN {X 0,Y 226.49,Z 557.296,A -85,B 0,C 180,E1 -21104.147,E2 -21104.147} C_VEL
LIN {X 0,Y 223.191,Z 566.13,A -85,B 0,C 180,E1 -21106.153,E2 -21106.153} C_VEL
LIN {X 0,Y 219.809,Z 574.151,A -85,B 0,C 180,E1 -21108.438,E2 -21108.438} C_VEL
LIN {X 0,Y 216.14,Z 582.005,A -85,B 0,C 180,E1 -21111.297,E2 -21111.297} C_VEL
LIN {X 0,Y 213.574,Z 587.121,A -85,B 0,C 180,E1 -21113.679,E2 -21113.679} C_VEL
LIN {X 0,Y 211.133,Z 591.623,A -85,B 0,C 180,E1 -21116.324,E2 -21116.324} C_VEL
LIN {X 0,Y 208.67,Z 595.824,A -85,B 0,C 180,E1 -21119.656,E2 -21119.656} C_VEL
LIN {X 0,Y 207.487,Z 597.722,A -85,B 0,C 180,E1 -21121.725,E2 -21121.725} C_VEL
LIN {X 0,Y 206.48,Z 599.068,A -85,B 0,C 180,E1 -21123.738,E2 -21123.738} C_VEL
LIN {X 0,Y 205.171,Z 600.495,A -85,B 0,C 180,E1 -21127.651,E2 -21127.651} C_VEL
LIN {X 0,Y 204.658,Z 600.586,A -85,B 0,C 180,E1 -21129.916,E2 -21129.916} C_VEL
LIN {X 0,Y 204.369,Z 600.229,A -85,B 0,C 180,E1 -21131.971,E2 -21131.971} C_VEL
LIN {X 0,Y 204.3,Z 599.269,A -85,B 0,C 180,E1 -21134.413,E2 -21134.413} C_VEL
LIN {X 0,Y 204.432,Z 596.61,A -85,B 0,C 180,E1 -21138.096,E2 -21138.096} C_VEL
LIN {X 0,Y 204.972,Z 593.303,A -85,B 0,C 180,E1 -21141.124,E2 -21141.124} C_VEL
LIN {X 0,Y 205.781,Z 588.908,A -85,B 0,C 180,E1 -21144.119,E2 -21144.119} C_VEL
LIN {X 0,Y 206.793,Z 583.323,A -85,B 0,C 180,E1 -21147.078,E2 -21147.078} C_VEL
LIN {X 0,Y 208.196,Z 576.352,A -85,B 0,C 180,E1 -21150,E2 -21150} C_VEL
LIN {X 0,Y 210.047,Z 567.598,A -85,B 0,C 180,E1 -21152.877,E2 -21152.877} C_VEL
LIN {X 0,Y 212.037,Z 558.027,A -85,B 0,C 180,E1 -21155.373,E2 -21155.373} C_VEL
LIN {X 0,Y 213.957,Z 547.557,A -85,B 0,C 180,E1 -21157.55,E2 -21157.55} C_VEL
LIN {X 0,Y 215.877,Z 536.309,A -85,B 0,C 180,E1 -21159.368,E2 -21159.368} C_VEL
LIN {X 0,Y 217.624,Z 523.729,A -85,B 0,C 180,E1 -21160.937,E2 -21160.937} C_VEL
LIN {X 0,Y 218.967,Z 510.793,A -85,B 0,C 180,E1 -21162.1,E2 -21162.1} C_VEL
LIN {X 0,Y 219.966,Z 496.975,A -85,B 0,C 180,E1 -21162.923,E2 -21162.923} C_VEL
LIN {X 0,Y 222.504,Z 431.436,A -85,B 0,C 180,E1 -21165.011,E2 -21165.011} C_VEL
LIN {X 0,Y 217.959,Z 419.166,A -85,B 0,C 180,E1 -21166.032,E2 -21166.032} C_VEL
LIN {X 0,Y 209.898,Z 402.203,A -85,B 0,C 180,E1 -21167.787,E2 -21167.787} C_VEL
LIN {X 0,Y 207.006,Z 396.629,A -85,B 0,C 180,E1 -21168.436,E2 -21168.436} C_VEL
LIN {X 0,Y 206.839,Z 395.721,A -85,B 0,C 180,E1 -21168.544,E2 -21168.544} C_VEL
LIN {X 0,Y 206.767,Z 395.716,A -85,B 0,C 180,E1 -21174.071,E2 -21174.071} C_VEL
LIN {X 0,Y 206.747,Z 395.731,A -85,B 0,C 180,E1 -21178.418,E2 -21178.418} C_VEL
LIN {X 0,Y 206.704,Z 395.735,A -85,B 0,C 180,E1 -21182.956,E2 -21182.956} C_VEL
LIN {X 0,Y 206.681,Z 395.738,A -85,B 0,C 180,E1 -21187.739,E2 -21187.739} C_VEL
LIN {X 0,Y 206.643,Z 395.738,A -85,B 0,C 180,E1 -21191.562,E2 -21191.562} C_VEL
LIN {X 0,Y 206.634,Z 395.74,A -85,B 0,C 180,E1 -21195.58,E2 -21195.58} C_VEL
LIN {X 0,Y 206.66,Z 395.74,A -85,B 0,C 180,E1 -21199.748,E2 -21199.748} C_VEL
LIN {X 0,Y 206.698,Z 395.735,A -85,B 0,C 180,E1 -21204.688,E2 -21204.688} C_VEL
LIN {X 0,Y 206.712,Z 395.728,A -85,B 0,C 180,E1 -21209.336,E2 -21209.336} C_VEL
LIN {X 0,Y 206.731,Z 395.732,A -85,B 0,C 180,E1 -21213.771,E2 -21213.771} C_VEL
LIN {X 0,Y 206.755,Z 395.725,A -85,B 0,C 180,E1 -21218.042,E2 -21218.042} C_VEL
LIN {X 0,Y 206.87,Z 395.712,A -85,B 0,C 180,E1 -21222.196,E2 -21222.196} C_VEL
LIN {X 0,Y 206.892,Z 395.71,A -85,B 0,C 180,E1 -21226.243,E2 -21226.243} C_VEL
LIN {X 0,Y 207.096,Z 395.68,A -85,B 0,C 180,E1 -21230.23,E2 -21230.23} C_VEL
LIN {X 0,Y 207.062,Z 395.69,A -85,B 0,C 180,E1 -21234.155,E2 -21234.155} C_VEL
LIN {X 0,Y 207.378,Z 395.64,A -85,B 0,C 180,E1 -21238.057,E2 -21238.057} C_VEL
LIN {X 0,Y 207.51,Z 395.607,A -85,B 0,C 180,E1 -21240,E2 -21240} C_VEL
LIN {X 0,Y 207.377,Z 395.617,A -85,B 0,C 180,E1 -21241.942,E2 -21241.942} C_VEL
LIN {X 0,Y 207.136,Z 395.681,A -85,B 0,C 180,E1 -21247.8,E2 -21247.8} C_VEL
LIN {X 0,Y 206.919,Z 395.702,A -85,B 0,C 180,E1 -21251.758,E2 -21251.758} C_VEL
LIN {X 0,Y 206.862,Z 395.717,A -85,B 0,C 180,E1 -21255.771,E2 -21255.771} C_VEL
LIN {X 0,Y 206.779,Z 395.725,A -85,B 0,C 180,E1 -21259.869,E2 -21259.869} C_VEL
LIN {X 0,Y 206.76,Z 395.727,A -85,B 0,C 180,E1 -21264.072,E2 -21264.072} C_VEL
LIN {X 0,Y 206.741,Z 395.731,A -85,B 0,C 180,E1 -21268.419,E2 -21268.419} C_VEL
LIN {X 0,Y 206.706,Z 395.739,A -85,B 0,C 180,E1 -21272.956,E2 -21272.956} C_VEL
LIN {X 0,Y 206.722,Z 395.74,A -85,B 0,C 180,E1 -21277.73,E2 -21277.73} C_VEL
LIN {X 0,Y 206.721,Z 395.74,A -85,B 0,C 180,E1 -21281.589,E2 -21281.589} C_VEL
LIN {X 0,Y 206.716,Z 395.739,A -85,B 0,C 180,E1 -21285.558,E2 -21285.558} C_VEL
LIN {X 0,Y 206.807,Z 395.812,A -85,B 0,C 180,E1 -21290.531,E2 -21290.531} C_VEL
LIN {X 0,Y 208.231,Z 402.092,A -85,B 0,C 180,E1 -21293.517,E2 -21293.517} C_VEL
LIN {X 0,Y 208.546,Z 404.545,A -85,B 0,C 180,E1 -21294.33,E2 -21294.33} C_VEL
LIN {X 0,Y 208.785,Z 409.423,A -85,B 0,C 180,E1 -21295.216,E2 -21295.216} C_VEL
LIN {X 0,Y 208.952,Z 414.992,A -85,B 0,C 180,E1 -21295.791,E2 -21295.791} C_VEL
LIN {X 0,Y 209.891,Z 425.102,A -85,B 0,C 180,E1 -21296.431,E2 -21296.431} C_VEL
LIN {X 0,Y 211.402,Z 430.919,A -85,B 0,C 180,E1 -21296.863,E2 -21296.863} C_VEL
LIN {X 0,Y 215.068,Z 465.404,A -85,B 0,C 180,E1 -21298.633,E2 -21298.633} C_VEL
LIN {X 0,Y 213.107,Z 515.116,A -85,B 0,C 180,E1 -21300.269,E2 -21300.269} C_VEL
LIN {X 0,Y 212.016,Z 528.631,A -85,B 0,C 180,E1 -21301.07,E2 -21301.07} C_VEL
LIN {X 0,Y 210.482,Z 540.796,A -85,B 0,C 180,E1 -21302.131,E2 -21302.131} C_VEL
LIN {X 0,Y 208.728,Z 552.29,A -85,B 0,C 180,E1 -21303.505,E2 -21303.505} C_VEL
LIN {X 0,Y 206.614,Z 562.74,A -85,B 0,C 180,E1 -21305.107,E2 -21305.107} C_VEL
LIN {X 0,Y 205.006,Z 571.422,A -85,B 0,C 180,E1 -21306.782,E2 -21306.782} C_VEL
LIN {X 0,Y 203.24,Z 580.088,A -85,B 0,C 180,E1 -21308.817,E2 -21308.817} C_VEL
LIN {X 0,Y 201.856,Z 586.795,A -85,B 0,C 180,E1 -21310.714,E2 -21310.714} C_VEL
LIN {X 0,Y 200.117,Z 595.422,A -85,B 0,C 180,E1 -21313.683,E2 -21313.683} C_VEL
LIN {X 0,Y 198.714,Z 602.358,A -85,B 0,C 180,E1 -21316.71,E2 -21316.71} C_VEL
LIN {X 0,Y 197.934,Z 607.909,A -85,B 0,C 180,E1 -21319.774,E2 -21319.774} C_VEL
LIN {X 0,Y 197.573,Z 612.236,A -85,B 0,C 180,E1 -21322.848,E2 -21322.848} C_VEL
LIN {X 0,Y 197.413,Z 615.451,A -85,B 0,C 180,E1 -21325.917,E2 -21325.917} C_VEL
LIN {X 0,Y 197.524,Z 617.043,A -85,B 0,C 180,E1 -21327.961,E2 -21327.961} C_VEL
LIN {X 0,Y 197.611,Z 618.208,A -85,B 0,C 180,E1 -21330,E2 -21330} C_VEL
LIN {X 0,Y 197.489,Z 618.906,A -85,B 0,C 180,E1 -21332.039,E2 -21332.039} C_VEL
LIN {X 0,Y 197.404,Z 619.231,A -85,B 0,C 180,E1 -21334.543,E2 -21334.543} C_VEL
LIN {X 0,Y 197.572,Z 618.663,A -85,B 0,C 180,E1 -21338.18,E2 -21338.18} C_VEL
LIN {X 0,Y 197.958,Z 617.787,A -85,B 0,C 180,E1 -21340.225,E2 -21340.225} C_VEL
LIN {X 0,Y 199.342,Z 614.835,A -85,B 0,C 180,E1 -21344.287,E2 -21344.287} C_VEL
LIN {X 0,Y 201.19,Z 611.521,A -85,B 0,C 180,E1 -21347.272,E2 -21347.272} C_VEL
LIN {X 0,Y 203.494,Z 607.17,A -85,B 0,C 180,E1 -21350.204,E2 -21350.204} C_VEL
LIN {X 0,Y 206.441,Z 601.385,A -85,B 0,C 180,E1 -21353.194,E2 -21353.194} C_VEL
LIN {X 0,Y 209.597,Z 594.832,A -85,B 0,C 180,E1 -21355.842,E2 -21355.842} C_VEL
LIN {X 0,Y 213.527,Z 586.356,A -85,B 0,C 180,E1 -21358.505,E2 -21358.505} C_VEL
LIN {X 0,Y 217.242,Z 577.673,A -85,B 0,C 180,E1 -21360.632,E2 -21360.632} C_VEL
LIN {X 0,Y 221.284,Z 567.019,A -85,B 0,C 180,E1 -21362.677,E2 -21362.677} C_VEL
LIN {X 0,Y 224.754,Z 556.457,A -85,B 0,C 180,E1 -21364.253,E2 -21364.253} C_VEL
LIN {X 0,Y 227.982,Z 544.699,A -85,B 0,C 180,E1 -21365.58,E2 -21365.58} C_VEL
LIN {X 0,Y 230.805,Z 531.267,A -85,B 0,C 180,E1 -21366.696,E2 -21366.696} C_VEL
LIN {X 0,Y 232.631,Z 519.106,A -85,B 0,C 180,E1 -21367.39,E2 -21367.39} C_VEL
LIN {X 0,Y 233.716,Z 506.319,A -85,B 0,C 180,E1 -21367.854,E2 -21367.854} C_VEL
LIN {X 0,Y 235.699,Z 471.709,A -85,B 0,C 180,E1 -21368.859,E2 -21368.859} C_VEL
LIN {X 0,Y 234.352,Z 460.876,A -85,B 0,C 180,E1 -21369.658,E2 -21369.658} C_VEL
LIN {X 0,Y 228.785,Z 448.145,A -85,B 0,C 180,E1 -21371.683,E2 -21371.683} C_VEL
LIN {X 0,Y 222.714,Z 435.926,A -85,B 0,C 180,E1 -21374.041,E2 -21374.041} C_VEL
LIN {X 0,Y 218.635,Z 428.886,A -85,B 0,C 180,E1 -21375.711,E2 -21375.711} C_VEL
LIN {X 0,Y 213.558,Z 420.509,A -85,B 0,C 180,E1 -21377.967,E2 -21377.967} C_VEL
LIN {X 0,Y 210.038,Z 414.993,A -85,B 0,C 180,E1 -21379.665,E2 -21379.665} C_VEL
LIN {X 0,Y 206.859,Z 410.289,A -85,B 0,C 180,E1 -21381.303,E2 -21381.303} C_VEL
LIN {X 0,Y 205.808,Z 408.829,A -85,B 0,C 180,E1 -21381.866,E2 -21381.866} C_VEL
LIN {X 0,Y 202.29,Z 404.127,A -85,B 0,C 180,E1 -21383.853,E2 -21383.853} C_VEL
LIN {X 0,Y 201.652,Z 402.853,A -85,B 0,C 180,E1 -21384.284,E2 -21384.284} C_VEL
LIN {X 0,Y 200.304,Z 398.753,A -85,B 0,C 180,E1 -21388.245,E2 -21388.245} C_VEL
LIN {X 0,Y 199.658,Z 396.603,A -85,B 0,C 180,E1 -21390.642,E2 -21390.642} C_VEL
LIN {X 0,Y 199.669,Z 396.603,A -85,B 0,C 180,E1 -21395.016,E2 -21395.016} C_VEL
LIN {X 0,Y 199.704,Z 396.599,A -85,B 0,C 180,E1 -21399.396,E2 -21399.396} C_VEL
LIN {X 0,Y 199.834,Z 396.582,A -85,B 0,C 180,E1 -21401.722,E2 -21401.722} C_VEL
LIN {X 0,Y 199.829,Z 396.59,A -85,B 0,C 180,E1 -21405.748,E2 -21405.748} C_VEL
LIN {X 0,Y 200.067,Z 396.565,A -85,B 0,C 180,E1 -21409.884,E2 -21409.884} C_VEL
LIN {X 0,Y 200.03,Z 396.558,A -85,B 0,C 180,E1 -21413.95,E2 -21413.95} C_VEL
LIN {X 0,Y 200.317,Z 396.516,A -85,B 0,C 180,E1 -21417.99,E2 -21417.99} C_VEL
LIN {X 0,Y 200.478,Z 396.514,A -85,B 0,C 180,E1 -21420,E2 -21420} C_VEL
LIN {X 0,Y 200.025,Z 396.561,A -85,B 0,C 180,E1 -21424.03,E2 -21424.03} C_VEL
LIN {X 0,Y 200.085,Z 396.548,A -85,B 0,C 180,E1 -21428.077,E2 -21428.077} C_VEL
LIN {X 0,Y 199.871,Z 396.574,A -85,B 0,C 180,E1 -21432.18,E2 -21432.18} C_VEL
LIN {X 0,Y 199.81,Z 396.583,A -85,B 0,C 180,E1 -21436.344,E2 -21436.344} C_VEL
LIN {X 0,Y 199.803,Z 396.766,A -85,B 0,C 180,E1 -21438.988,E2 -21438.988} C_VEL
LIN {X 0,Y 200.673,Z 399.277,A -85,B 0,C 180,E1 -21439.651,E2 -21439.651} C_VEL
LIN {X 0,Y 202.511,Z 401.399,A -85,B 0,C 180,E1 -21440.745,E2 -21440.745} C_VEL
LIN {X 0,Y 204.164,Z 402.527,A -85,B 0,C 180,E1 -21441.629,E2 -21441.629} C_VEL
LIN {X 0,Y 206.104,Z 405.745,A -85,B 0,C 180,E1 -21442.745,E2 -21442.745} C_VEL
LIN {X 0,Y 208.355,Z 407.964,A -85,B 0,C 180,E1 -21443.877,E2 -21443.877} C_VEL
LIN {X 0,Y 210.838,Z 411.448,A -85,B 0,C 180,E1 -21445.123,E2 -21445.123} C_VEL
LIN {X 0,Y 212.108,Z 412.955,A -85,B 0,C 180,E1 -21445.717,E2 -21445.717} C_VEL
LIN {X 0,Y 214.917,Z 416.706,A -85,B 0,C 180,E1 -21447.002,E2 -21447.002} C_VEL
LIN {X 0,Y 221.617,Z 426.211,A -85,B 0,C 180,E1 -21449.809,E2 -21449.809} C_VEL
LIN {X 0,Y 228.224,Z 436.456,A -85,B 0,C 180,E1 -21452.299,E2 -21452.299} C_VEL
LIN {X 0,Y 232.612,Z 444.428,A -85,B 0,C 180,E1 -21453.858,E2 -21453.858} C_VEL
LIN {X 0,Y 236.669,Z 453.113,A -85,B 0,C 180,E1 -21455.263,E2 -21455.263} C_VEL
LIN {X 0,Y 233.958,Z 498.807,A -85,B 0,C 180,E1 -21456.643,E2 -21456.643} C_VEL
LIN {X 0,Y 232.31,Z 512.493,A -85,B 0,C 180,E1 -21457.376,E2 -21457.376} C_VEL
LIN {X 0,Y 230.174,Z 524.622,A -85,B 0,C 180,E1 -21458.343,E2 -21458.343} C_VEL
LIN {X 0,Y 227.721,Z 535.385,A -85,B 0,C 180,E1 -21459.508,E2 -21459.508} C_VEL
LIN {X 0,Y 224.523,Z 546.692,A -85,B 0,C 180,E1 -21461.098,E2 -21461.098} C_VEL
LIN {X 0,Y 220.916,Z 557.171,A -85,B 0,C 180,E1 -21462.972,E2 -21462.972} C_VEL
LIN {X 0,Y 217.015,Z 567.117,A -85,B 0,C 180,E1 -21465.281,E2 -21465.281} C_VEL
LIN {X 0,Y 212.881,Z 576.315,A -85,B 0,C 180,E1 -21468.048,E2 -21468.048} C_VEL
LIN {X 0,Y 209.189,Z 583.717,A -85,B 0,C 180,E1 -21470.956,E2 -21470.956} C_VEL
LIN {X 0,Y 206.54,Z 588.668,A -85,B 0,C 180,E1 -21473.454,E2 -21473.454} C_VEL
LIN {X 0,Y 203.762,Z 593.347,A -85,B 0,C 180,E1 -21476.506,E2 -21476.506} C_VEL
LIN {X 0,Y 202.192,Z 595.775,A -85,B 0,C 180,E1 -21478.576,E2 -21478.576} C_VEL
LIN {X 0,Y 200.644,Z 598.094,A -85,B 0,C 180,E1 -21481.127,E2 -21481.127} C_VEL
LIN {X 0,Y 198.894,Z 600.212,A -85,B 0,C 180,E1 -21484.912,E2 -21484.912} C_VEL
LIN {X 0,Y 198.171,Z 600.84,A -85,B 0,C 180,E1 -21487.233,E2 -21487.233} C_VEL
LIN {X 0,Y 197.698,Z 600.961,A -85,B 0,C 180,E1 -21489.177,E2 -21489.177} C_VEL
LIN {X 0,Y 197.343,Z 600.663,A -85,B 0,C 180,E1 -21491.306,E2 -21491.306} C_VEL
LIN {X 0,Y 197.201,Z 599.611,A -85,B 0,C 180,E1 -21494.209,E2 -21494.209} C_VEL
LIN {X 0,Y 197.286,Z 597.279,A -85,B 0,C 180,E1 -21497.659,E2 -21497.659} C_VEL
LIN {X 0,Y 197.81,Z 594.095,A -85,B 0,C 180,E1 -21500.8,E2 -21500.8} C_VEL
LIN {X 0,Y 198.595,Z 589.834,A -85,B 0,C 180,E1 -21503.906,E2 -21503.906} C_VEL
LIN {X 0,Y 199.818,Z 583.367,A -85,B 0,C 180,E1 -21507.48,E2 -21507.48} C_VEL
LIN {X 0,Y 201.313,Z 576.315,A -85,B 0,C 180,E1 -21510.5,E2 -21510.5} C_VEL
LIN {X 0,Y 203.263,Z 567.459,A -85,B 0,C 180,E1 -21513.469,E2 -21513.469} C_VEL
LIN {X 0,Y 205.427,Z 557.399,A -85,B 0,C 180,E1 -21516.137,E2 -21516.137} C_VEL
LIN {X 0,Y 207.352,Z 547.142,A -85,B 0,C 180,E1 -21518.282,E2 -21518.282} C_VEL
LIN {X 0,Y 209.374,Z 535.719,A -85,B 0,C 180,E1 -21520.15,E2 -21520.15} C_VEL
LIN {X 0,Y 211.043,Z 523.904,A -85,B 0,C 180,E1 -21521.647,E2 -21521.647} C_VEL
LIN {X 0,Y 212.401,Z 511.626,A -85,B 0,C 180,E1 -21522.784,E2 -21522.784} C_VEL
LIN {X 0,Y 213.417,Z 498.099,A -85,B 0,C 180,E1 -21523.629,E2 -21523.629} C_VEL
LIN {X 0,Y 215.442,Z 450.909,A -85,B 0,C 180,E1 -21525.188,E2 -21525.188} C_VEL
LIN {X 0,Y 216.104,Z 433.156,A -85,B 0,C 180,E1 -21525.758,E2 -21525.758} C_VEL
LIN {X 0,Y 212.244,Z 422.67,A -85,B 0,C 180,E1 -21526.669,E2 -21526.669} C_VEL
LIN {X 0,Y 204.371,Z 405.958,A -85,B 0,C 180,E1 -21528.469,E2 -21528.469} C_VEL
LIN {X 0,Y 200.04,Z 397.852,A -85,B 0,C 180,E1 -21529.488,E2 -21529.488} C_VEL
LIN {X 0,Y 199.761,Z 396.603,A -85,B 0,C 180,E1 -21529.613,E2 -21529.613} C_VEL
LIN {X 0,Y 199.74,Z 396.591,A -85,B 0,C 180,E1 -21533.816,E2 -21533.816} C_VEL
LIN {X 0,Y 199.715,Z 396.607,A -85,B 0,C 180,E1 -21538.386,E2 -21538.386} C_VEL
LIN {X 0,Y 199.679,Z 396.609,A -85,B 0,C 180,E1 -21542.357,E2 -21542.357} C_VEL
LIN {X 0,Y 199.624,Z 396.614,A -85,B 0,C 180,E1 -21546.762,E2 -21546.762} C_VEL
LIN {X 0,Y 199.609,Z 396.62,A -85,B 0,C 180,E1 -21549.327,E2 -21549.327} C_VEL
LIN {X 0,Y 199.575,Z 396.618,A -85,B 0,C 180,E1 -21552.309,E2 -21552.309} C_VEL
LIN {X 0,Y 199.581,Z 396.62,A -85,B 0,C 180,E1 -21555.228,E2 -21555.228} C_VEL
LIN {X 0,Y 199.58,Z 396.619,A -85,B 0,C 180,E1 -21558.004,E2 -21558.004} C_VEL
LIN {X 0,Y 199.61,Z 396.619,A -85,B 0,C 180,E1 -21560.766,E2 -21560.766} C_VEL
LIN {X 0,Y 199.611,Z 396.619,A -85,B 0,C 180,E1 -21565.712,E2 -21565.712} C_VEL
LIN {X 0,Y 199.692,Z 396.607,A -85,B 0,C 180,E1 -21568.135,E2 -21568.135} C_VEL
LIN {X 0,Y 199.685,Z 396.612,A -85,B 0,C 180,E1 -21572.771,E2 -21572.771} C_VEL
LIN {X 0,Y 199.735,Z 396.599,A -85,B 0,C 180,E1 -21577.228,E2 -21577.228} C_VEL
LIN {X 0,Y 199.794,Z 396.593,A -85,B 0,C 180,E1 -21581.757,E2 -21581.757} C_VEL
LIN {X 0,Y 199.832,Z 396.588,A -85,B 0,C 180,E1 -21585.747,E2 -21585.747} C_VEL
LIN {X 0,Y 200.019,Z 396.562,A -85,B 0,C 180,E1 -21589.881,E2 -21589.881} C_VEL
LIN {X 0,Y 200.023,Z 396.566,A -85,B 0,C 180,E1 -21593.949,E2 -21593.949} C_VEL
LIN {X 0,Y 200.317,Z 396.519,A -85,B 0,C 180,E1 -21597.989,E2 -21597.989} C_VEL
LIN {X 0,Y 200.475,Z 396.482,A -85,B 0,C 180,E1 -21600,E2 -21600} C_VEL
LIN {X 0,Y 200.022,Z 396.55,A -85,B 0,C 180,E1 -21604.029,E2 -21604.029} C_VEL
LIN {X 0,Y 200.084,Z 396.561,A -85,B 0,C 180,E1 -21608.076,E2 -21608.076} C_VEL
LIN {X 0,Y 199.87,Z 396.581,A -85,B 0,C 180,E1 -21612.179,E2 -21612.179} C_VEL
LIN {X 0,Y 199.8,Z 396.595,A -85,B 0,C 180,E1 -21616.343,E2 -21616.343} C_VEL
LIN {X 0,Y 199.696,Z 396.611,A -85,B 0,C 180,E1 -21620.605,E2 -21620.605} C_VEL
LIN {X 0,Y 199.669,Z 396.613,A -85,B 0,C 180,E1 -21624.984,E2 -21624.984} C_VEL
LIN {X 0,Y 199.672,Z 396.613,A -85,B 0,C 180,E1 -21629.522,E2 -21629.522} C_VEL
LIN {X 0,Y 199.661,Z 396.615,A -85,B 0,C 180,E1 -21632.352,E2 -21632.352} C_VEL
LIN {X 0,Y 199.65,Z 396.62,A -85,B 0,C 180,E1 -21636.757,E2 -21636.757} C_VEL
LIN {X 0,Y 199.676,Z 396.618,A -85,B 0,C 180,E1 -21639.312,E2 -21639.312} C_VEL
LIN {X 0,Y 199.66,Z 396.62,A -85,B 0,C 180,E1 -21642.339,E2 -21642.339} C_VEL
LIN {X 0,Y 199.663,Z 396.618,A -85,B 0,C 180,E1 -21645.254,E2 -21645.254} C_VEL
LIN {X 0,Y 199.757,Z 396.665,A -85,B 0,C 180,E1 -21649.762,E2 -21649.762} C_VEL
LIN {X 0,Y 201.912,Z 406.355,A -85,B 0,C 180,E1 -21654.503,E2 -21654.503} C_VEL
LIN {X 0,Y 209.91,Z 426.823,A -85,B 0,C 180,E1 -21656.5,E2 -21656.5} C_VEL
LIN {X 0,Y 211.402,Z 430.919,A -85,B 0,C 180,E1 -21656.863,E2 -21656.863} C_VEL
LIN {X 0,Y 212.214,Z 434.577,A -85,B 0,C 180,E1 -21657.112,E2 -21657.112} C_VEL
LIN {X 0,Y 211.997,Z 440.391,A -85,B 0,C 180,E1 -21657.303,E2 -21657.303} C_VEL
LIN {X 0,Y 208.48,Z 456.187,A -85,B 0,C 180,E1 -21657.43,E2 -21657.43} C_VEL
LIN {X 0,Y 208.265,Z 462.194,A -85,B 0,C 180,E1 -21657.631,E2 -21657.631} C_VEL
LIN {X 0,Y 208.595,Z 467.961,A -85,B 0,C 180,E1 -21657.896,E2 -21657.896} C_VEL
LIN {X 0,Y 206.653,Z 514.636,A -85,B 0,C 180,E1 -21659.47,E2 -21659.47} C_VEL
LIN {X 0,Y 205.509,Z 528.025,A -85,B 0,C 180,E1 -21660.274,E2 -21660.274} C_VEL
LIN {X 0,Y 203.874,Z 540.841,A -85,B 0,C 180,E1 -21661.426,E2 -21661.426} C_VEL
LIN {X 0,Y 202.06,Z 552.23,A -85,B 0,C 180,E1 -21662.838,E2 -21662.838} C_VEL
LIN {X 0,Y 199.871,Z 562.623,A -85,B 0,C 180,E1 -21664.486,E2 -21664.486} C_VEL
LIN {X 0,Y 198.21,Z 571.273,A -85,B 0,C 180,E1 -21666.214,E2 -21666.214} C_VEL
LIN {X 0,Y 196.236,Z 580.449,A -85,B 0,C 180,E1 -21668.464,E2 -21668.464} C_VEL
LIN {X 0,Y 194.961,Z 586.217,A -85,B 0,C 180,E1 -21670.153,E2 -21670.153} C_VEL
LIN {X 0,Y 193.258,Z 594.562,A -85,B 0,C 180,E1 -21673.087,E2 -21673.087} C_VEL
LIN {X 0,Y 191.753,Z 601.602,A -85,B 0,C 180,E1 -21676.218,E2 -21676.218} C_VEL
LIN {X 0,Y 190.923,Z 607.241,A -85,B 0,C 180,E1 -21679.394,E2 -21679.394} C_VEL
LIN {X 0,Y 190.495,Z 611.645,A -85,B 0,C 180,E1 -21682.581,E2 -21682.581} C_VEL
LIN {X 0,Y 190.323,Z 614.933,A -85,B 0,C 180,E1 -21685.765,E2 -21685.765} C_VEL
LIN {X 0,Y 190.436,Z 616.56,A -85,B 0,C 180,E1 -21687.885,E2 -21687.885} C_VEL
LIN {X 0,Y 190.546,Z 617.767,A -85,B 0,C 180,E1 -21690,E2 -21690} C_VEL
LIN {X 0,Y 190.404,Z 618.521,A -85,B 0,C 180,E1 -21692.115,E2 -21692.115} C_VEL
LIN {X 0,Y 190.329,Z 618.866,A -85,B 0,C 180,E1 -21694.45,E2 -21694.45} C_VEL
LIN {X 0,Y 190.519,Z 618.377,A -85,B 0,C 180,E1 -21698.485,E2 -21698.485} C_VEL
LIN {X 0,Y 190.956,Z 617.563,A -85,B 0,C 180,E1 -21700.604,E2 -21700.604} C_VEL
LIN {X 0,Y 192.435,Z 614.683,A -85,B 0,C 180,E1 -21704.812,E2 -21704.812} C_VEL
LIN {X 0,Y 194.405,Z 611.443,A -85,B 0,C 180,E1 -21707.895,E2 -21707.895} C_VEL
LIN {X 0,Y 196.837,Z 607.168,A -85,B 0,C 180,E1 -21710.918,E2 -21710.918} C_VEL
LIN {X 0,Y 200.26,Z 600.841,A -85,B 0,C 180,E1 -21714.295,E2 -21714.295} C_VEL
LIN {X 0,Y 203.864,Z 593.77,A -85,B 0,C 180,E1 -21717.179,E2 -21717.179} C_VEL
LIN {X 0,Y 208.097,Z 585.084,A -85,B 0,C 180,E1 -21719.877,E2 -21719.877} C_VEL
LIN {X 0,Y 211.967,Z 576.228,A -85,B 0,C 180,E1 -21722.038,E2 -21722.038} C_VEL
LIN {X 0,Y 216.206,Z 565.352,A -85,B 0,C 180,E1 -21724.105,E2 -21724.105} C_VEL
LIN {X 0,Y 219.918,Z 554.375,A -85,B 0,C 180,E1 -21725.676,E2 -21725.676} C_VEL
LIN {X 0,Y 223.248,Z 542.134,A -85,B 0,C 180,E1 -21727.017,E2 -21727.017} C_VEL
LIN {X 0,Y 225.702,Z 530.591,A -85,B 0,C 180,E1 -21727.95,E2 -21727.95} C_VEL
LIN {X 0,Y 227.698,Z 517.478,A -85,B 0,C 180,E1 -21728.673,E2 -21728.673} C_VEL
LIN {X 0,Y 229.021,Z 500.373,A -85,B 0,C 180,E1 -21729.249,E2 -21729.249} C_VEL
LIN {X 0,Y 230.606,Z 472.408,A -85,B 0,C 180,E1 -21730.094,E2 -21730.094} C_VEL
LIN {X 0,Y 229.569,Z 464.041,A -85,B 0,C 180,E1 -21730.741,E2 -21730.741} C_VEL
LIN {X 0,Y 224.698,Z 452.604,A -85,B 0,C 180,E1 -21732.624,E2 -21732.624} C_VEL
LIN {X 0,Y 218.962,Z 440.797,A -85,B 0,C 180,E1 -21734.976,E2 -21734.976} C_VEL
LIN {X 0,Y 213.768,Z 431.522,A -85,B 0,C 180,E1 -21737.262,E2 -21737.262} C_VEL
LIN {X 0,Y 209.876,Z 425.189,A -85,B 0,C 180,E1 -21739.114,E2 -21739.114} C_VEL
LIN {X 0,Y 207.11,Z 420.686,A -85,B 0,C 180,E1 -21740.531,E2 -21740.531} C_VEL
LIN {X 0,Y 203.876,Z 415.663,A -85,B 0,C 180,E1 -21742.295,E2 -21742.295} C_VEL
LIN {X 0,Y 199.866,Z 410.237,A -85,B 0,C 180,E1 -21744.643,E2 -21744.643} C_VEL
LIN {X 0,Y 198.699,Z 408.46,A -85,B 0,C 180,E1 -21745.394,E2 -21745.394} C_VEL
LIN {X 0,Y 195.212,Z 404.056,A -85,B 0,C 180,E1 -21747.773,E2 -21747.773} C_VEL
LIN {X 0,Y 194.054,Z 401.967,A -85,B 0,C 180,E1 -21748.779,E2 -21748.779} C_VEL
LIN {X 0,Y 193.166,Z 399.38,A -85,B 0,C 180,E1 -21751.772,E2 -21751.772} C_VEL
LIN {X 0,Y 192.595,Z 397.481,A -85,B 0,C 180,E1 -21754.277,E2 -21754.277} C_VEL
LIN {X 0,Y 192.702,Z 397.48,A -85,B 0,C 180,E1 -21756.349,E2 -21756.349} C_VEL
LIN {X 0,Y 192.778,Z 397.464,A -85,B 0,C 180,E1 -21761.414,E2 -21761.414} C_VEL
LIN {X 0,Y 192.758,Z 397.476,A -85,B 0,C 180,E1 -21765.214,E2 -21765.214} C_VEL
LIN {X 0,Y 192.978,Z 397.444,A -85,B 0,C 180,E1 -21769.509,E2 -21769.509} C_VEL
LIN {X 0,Y 193.057,Z 397.423,A -85,B 0,C 180,E1 -21771.628,E2 -21771.628} C_VEL
LIN {X 0,Y 193.259,Z 397.395,A -85,B 0,C 180,E1 -21777.916,E2 -21777.916} C_VEL
LIN {X 0,Y 193.442,Z 397.39,A -85,B 0,C 180,E1 -21780.001,E2 -21780.001} C_VEL
LIN {X 0,Y 192.971,Z 397.44,A -85,B 0,C 180,E1 -21784.178,E2 -21784.178} C_VEL
LIN {X 0,Y 193.033,Z 397.428,A -85,B 0,C 180,E1 -21788.375,E2 -21788.375} C_VEL
LIN {X 0,Y 192.799,Z 397.456,A -85,B 0,C 180,E1 -21792.634,E2 -21792.634} C_VEL
LIN {X 0,Y 192.769,Z 397.47,A -85,B 0,C 180,E1 -21794.719,E2 -21794.719} C_VEL
LIN {X 0,Y 193.522,Z 399.926,A -85,B 0,C 180,E1 -21795.468,E2 -21795.468} C_VEL
LIN {X 0,Y 195.432,Z 402.159,A -85,B 0,C 180,E1 -21796.887,E2 -21796.887} C_VEL
LIN {X 0,Y 197.418,Z 403.43,A -85,B 0,C 180,E1 -21798.176,E2 -21798.176} C_VEL
LIN {X 0,Y 199.055,Z 406.454,A -85,B 0,C 180,E1 -21799.33,E2 -21799.33} C_VEL
LIN {X 0,Y 201.87,Z 409.104,A -85,B 0,C 180,E1 -21800.974,E2 -21800.974} C_VEL
LIN {X 0,Y 204.078,Z 412.403,A -85,B 0,C 180,E1 -21802.261,E2 -21802.261} C_VEL
LIN {X 0,Y 205.821,Z 414.271,A -85,B 0,C 180,E1 -21803.177,E2 -21803.177} C_VEL
LIN {X 0,Y 208.656,Z 417.993,A -85,B 0,C 180,E1 -21804.631,E2 -21804.631} C_VEL
LIN {X 0,Y 215.327,Z 427.273,A -85,B 0,C 180,E1 -21807.746,E2 -21807.746} C_VEL
LIN {X 0,Y 222.124,Z 437.552,A -85,B 0,C 180,E1 -21810.546,E2 -21810.546} C_VEL
LIN {X 0,Y 227.304,Z 446.592,A -85,B 0,C 180,E1 -21812.52,E2 -21812.52} C_VEL
LIN {X 0,Y 231.541,Z 455.498,A -85,B 0,C 180,E1 -21814.076,E2 -21814.076} C_VEL
LIN {X 0,Y 229.583,Z 488.982,A -85,B 0,C 180,E1 -21815.073,E2 -21815.073} C_VEL
LIN {X 0,Y 228.481,Z 503.351,A -85,B 0,C 180,E1 -21815.616,E2 -21815.616} C_VEL
LIN {X 0,Y 226.574,Z 516.542,A -85,B 0,C 180,E1 -21816.436,E2 -21816.436} C_VEL
LIN {X 0,Y 223.915,Z 529.402,A -85,B 0,C 180,E1 -21817.58,E2 -21817.58} C_VEL
LIN {X 0,Y 221.203,Z 540.08,A -85,B 0,C 180,E1 -21818.887,E2 -21818.887} C_VEL
LIN {X 0,Y 217.489,Z 551.552,A -85,B 0,C 180,E1 -21820.687,E2 -21820.687} C_VEL
LIN {X 0,Y 213.847,Z 561.302,A -85,B 0,C 180,E1 -21822.665,E2 -21822.665} C_VEL
LIN {X 0,Y 210.361,Z 569.361,A -85,B 0,C 180,E1 -21824.703,E2 -21824.703} C_VEL
LIN {X 0,Y 206.659,Z 577.08,A -85,B 0,C 180,E1 -21827.146,E2 -21827.146} C_VEL
LIN {X 0,Y 203.711,Z 582.706,A -85,B 0,C 180,E1 -21829.377,E2 -21829.377} C_VEL
LIN {X 0,Y 200.531,Z 588.346,A -85,B 0,C 180,E1 -21832.171,E2 -21832.171} C_VEL
LIN {X 0,Y 197.519,Z 593.194,A -85,B 0,C 180,E1 -21835.299,E2 -21835.299} C_VEL
LIN {X 0,Y 195.057,Z 596.819,A -85,B 0,C 180,E1 -21838.505,E2 -21838.505} C_VEL
LIN {X 0,Y 193.155,Z 599.328,A -85,B 0,C 180,E1 -21841.771,E2 -21841.771} C_VEL
LIN {X 0,Y 192.136,Z 600.412,A -85,B 0,C 180,E1 -21843.964,E2 -21843.964} C_VEL
LIN {X 0,Y 191.177,Z 601.185,A -85,B 0,C 180,E1 -21846.789,E2 -21846.789} C_VEL
LIN {X 0,Y 190.348,Z 601.097,A -85,B 0,C 180,E1 -21850.592,E2 -21850.592} C_VEL
LIN {X 0,Y 190.109,Z 599.954,A -85,B 0,C 180,E1 -21853.985,E2 -21853.985} C_VEL
LIN {X 0,Y 190.164,Z 597.94,A -85,B 0,C 180,E1 -21857.189,E2 -21857.189} C_VEL
LIN {X 0,Y 190.644,Z 594.877,A -85,B 0,C 180,E1 -21860.451,E2 -21860.451} C_VEL
LIN {X 0,Y 191.418,Z 590.747,A -85,B 0,C 180,E1 -21863.676,E2 -21863.676} C_VEL
LIN {X 0,Y 192.662,Z 584.419,A -85,B 0,C 180,E1 -21867.387,E2 -21867.387} C_VEL
LIN {X 0,Y 194.158,Z 577.539,A -85,B 0,C 180,E1 -21870.518,E2 -21870.518} C_VEL
LIN {X 0,Y 195.763,Z 570.513,A -85,B 0,C 180,E1 -21873.087,E2 -21873.087} C_VEL
LIN {X 0,Y 197.769,Z 561.671,A -85,B 0,C 180,E1 -21875.711,E2 -21875.711} C_VEL
LIN {X 0,Y 199.865,Z 551.596,A -85,B 0,C 180,E1 -21878.086,E2 -21878.086} C_VEL
LIN {X 0,Y 202.08,Z 539.812,A -85,B 0,C 180,E1 -21880.267,E2 -21880.267} C_VEL
LIN {X 0,Y 203.982,Z 528.02,A -85,B 0,C 180,E1 -21881.93,E2 -21881.93} C_VEL
LIN {X 0,Y 205.529,Z 515.782,A -85,B 0,C 180,E1 -21883.219,E2 -21883.219} C_VEL
LIN {X 0,Y 206.655,Z 503.2,A -85,B 0,C 180,E1 -21884.159,E2 -21884.159} C_VEL
LIN {X 0,Y 207.364,Z 490.543,A -85,B 0,C 180,E1 -21884.738,E2 -21884.738} C_VEL
LIN {X 0,Y 209.632,Z 434.373,A -85,B 0,C 180,E1 -21886.584,E2 -21886.584} C_VEL
LIN {X 0,Y 205.553,Z 423.824,A -85,B 0,C 180,E1 -21887.58,E2 -21887.58} C_VEL
LIN {X 0,Y 198.841,Z 409.659,A -85,B 0,C 180,E1 -21889.195,E2 -21889.195} C_VEL
LIN {X 0,Y 192.883,Z 398.58,A -85,B 0,C 180,E1 -21890.672,E2 -21890.672} C_VEL
LIN {X 0,Y 192.666,Z 397.486,A -85,B 0,C 180,E1 -21890.781,E2 -21890.781} C_VEL
LIN {X 0,Y 192.667,Z 397.472,A -85,B 0,C 180,E1 -21894.224,E2 -21894.224} C_VEL
LIN {X 0,Y 192.652,Z 397.486,A -85,B 0,C 180,E1 -21898.891,E2 -21898.891} C_VEL
LIN {X 0,Y 192.601,Z 397.492,A -85,B 0,C 180,E1 -21903.185,E2 -21903.185} C_VEL
LIN {X 0,Y 192.552,Z 397.497,A -85,B 0,C 180,E1 -21908.351,E2 -21908.351} C_VEL
LIN {X 0,Y 192.492,Z 397.504,A -85,B 0,C 180,E1 -21913.095,E2 -21913.095} C_VEL
LIN {X 0,Y 192.492,Z 397.499,A -85,B 0,C 180,E1 -21916.903,E2 -21916.903} C_VEL
LIN {X 0,Y 192.55,Z 397.494,A -85,B 0,C 180,E1 -21921.647,E2 -21921.647} C_VEL
LIN {X 0,Y 192.595,Z 397.495,A -85,B 0,C 180,E1 -21926.813,E2 -21926.813} C_VEL
LIN {X 0,Y 192.663,Z 397.484,A -85,B 0,C 180,E1 -21931.691,E2 -21931.691} C_VEL
LIN {X 0,Y 192.703,Z 397.471,A -85,B 0,C 180,E1 -21936.348,E2 -21936.348} C_VEL
LIN {X 0,Y 192.729,Z 397.473,A -85,B 0,C 180,E1 -21941.457,E2 -21941.457} C_VEL
LIN {X 0,Y 192.76,Z 397.47,A -85,B 0,C 180,E1 -21945.213,E2 -21945.213} C_VEL
LIN {X 0,Y 192.942,Z 397.443,A -85,B 0,C 180,E1 -21949.566,E2 -21949.566} C_VEL
LIN {X 0,Y 193.037,Z 397.43,A -85,B 0,C 180,E1 -21951.626,E2 -21951.626} C_VEL
LIN {X 0,Y 193.259,Z 397.398,A -85,B 0,C 180,E1 -21957.915,E2 -21957.915} C_VEL
LIN {X 0,Y 193.439,Z 397.356,A -85,B 0,C 180,E1 -21959.999,E2 -21959.999} C_VEL
LIN {X 0,Y 192.968,Z 397.428,A -85,B 0,C 180,E1 -21964.177,E2 -21964.177} C_VEL
LIN {X 0,Y 193.032,Z 397.441,A -85,B 0,C 180,E1 -21968.374,E2 -21968.374} C_VEL
LIN {X 0,Y 192.797,Z 397.464,A -85,B 0,C 180,E1 -21972.633,E2 -21972.633} C_VEL
LIN {X 0,Y 192.753,Z 397.469,A -85,B 0,C 180,E1 -21976.959,E2 -21976.959} C_VEL
LIN {X 0,Y 192.633,Z 397.489,A -85,B 0,C 180,E1 -21981.397,E2 -21981.397} C_VEL
LIN {X 0,Y 192.661,Z 397.483,A -85,B 0,C 180,E1 -21984.225,E2 -21984.225} C_VEL
LIN {X 0,Y 192.647,Z 397.489,A -85,B 0,C 180,E1 -21988.892,E2 -21988.892} C_VEL
LIN {X 0,Y 192.597,Z 397.496,A -85,B 0,C 180,E1 -21993.186,E2 -21993.186} C_VEL
LIN {X 0,Y 192.598,Z 397.5,A -85,B 0,C 180,E1 -21998.341,E2 -21998.341} C_VEL
LIN {X 0,Y 192.602,Z 397.498,A -85,B 0,C 180,E1 -22003.132,E2 -22003.132} C_VEL
LIN {X 0,Y 192.621,Z 397.492,A -85,B 0,C 180,E1 -22008.252,E2 -22008.252} C_VEL
LIN {X 0,Y 192.651,Z 397.567,A -85,B 0,C 180,E1 -22008.956,E2 -22008.956} C_VEL
LIN {X 0,Y 194.665,Z 406.093,A -85,B 0,C 180,E1 -22013.296,E2 -22013.296} C_VEL
LIN {X 0,Y 202.428,Z 425.365,A -85,B 0,C 180,E1 -22015.351,E2 -22015.351} C_VEL
LIN {X 0,Y 205.309,Z 433.367,A -85,B 0,C 180,E1 -22016.098,E2 -22016.098} C_VEL
LIN {X 0,Y 208.265,Z 462.194,A -85,B 0,C 180,E1 -22017.631,E2 -22017.631} C_VEL
LIN {X 0,Y 208.27,Z 466.067,A -85,B 0,C 180,E1 -22017.78,E2 -22017.78} C_VEL
LIN {X 0,Y 207.657,Z 469.937,A -85,B 0,C 180,E1 -22017.846,E2 -22017.846} C_VEL
LIN {X 0,Y 205.346,Z 477.538,A -85,B 0,C 180,E1 -22017.829,E2 -22017.829} C_VEL
LIN {X 0,Y 202.188,Z 487.095,A -85,B 0,C 180,E1 -22017.772,E2 -22017.772} C_VEL
LIN {X 0,Y 201.243,Z 492.996,A -85,B 0,C 180,E1 -22017.874,E2 -22017.874} C_VEL
LIN {X 0,Y 200.084,Z 516.202,A -85,B 0,C 180,E1 -22018.723,E2 -22018.723} C_VEL
LIN {X 0,Y 198.852,Z 529.746,A -85,B 0,C 180,E1 -22019.613,E2 -22019.613} C_VEL
LIN {X 0,Y 197.161,Z 541.938,A -85,B 0,C 180,E1 -22020.798,E2 -22020.798} C_VEL
LIN {X 0,Y 195.124,Z 553.764,A -85,B 0,C 180,E1 -22022.372,E2 -22022.372} C_VEL
LIN {X 0,Y 192.939,Z 563.827,A -85,B 0,C 180,E1 -22024.081,E2 -22024.081} C_VEL
LIN {X 0,Y 190.748,Z 574.382,A -85,B 0,C 180,E1 -22026.38,E2 -22026.38} C_VEL
LIN {X 0,Y 188.583,Z 583.343,A -85,B 0,C 180,E1 -22028.818,E2 -22028.818} C_VEL
LIN {X 0,Y 186.985,Z 590.898,A -85,B 0,C 180,E1 -22031.369,E2 -22031.369} C_VEL
LIN {X 0,Y 185.306,Z 598.606,A -85,B 0,C 180,E1 -22034.605,E2 -22034.605} C_VEL
LIN {X 0,Y 184.155,Z 604.789,A -85,B 0,C 180,E1 -22037.884,E2 -22037.884} C_VEL
LIN {X 0,Y 183.548,Z 609.677,A -85,B 0,C 180,E1 -22041.19,E2 -22041.19} C_VEL
LIN {X 0,Y 183.266,Z 613.399,A -85,B 0,C 180,E1 -22044.499,E2 -22044.499} C_VEL
LIN {X 0,Y 183.35,Z 616.075,A -85,B 0,C 180,E1 -22047.803,E2 -22047.803} C_VEL
LIN {X 0,Y 183.481,Z 617.317,A -85,B 0,C 180,E1 -22050,E2 -22050} C_VEL
LIN {X 0,Y 183.321,Z 618.129,A -85,B 0,C 180,E1 -22052.197,E2 -22052.197} C_VEL
LIN {X 0,Y 183.234,Z 618.503,A -85,B 0,C 180,E1 -22054.399,E2 -22054.399} C_VEL
LIN {X 0,Y 183.488,Z 618.091,A -85,B 0,C 180,E1 -22058.813,E2 -22058.813} C_VEL
LIN {X 0,Y 183.943,Z 617.319,A -85,B 0,C 180,E1 -22061.013,E2 -22061.013} C_VEL
LIN {X 0,Y 184.636,Z 616.135,A -85,B 0,C 180,E1 -22063.202,E2 -22063.202} C_VEL
LIN {X 0,Y 186.188,Z 613.609,A -85,B 0,C 180,E1 -22066.445,E2 -22066.445} C_VEL
LIN {X 0,Y 188.432,Z 610.106,A -85,B 0,C 180,E1 -22069.613,E2 -22069.613} C_VEL
LIN {X 0,Y 191.234,Z 605.549,A -85,B 0,C 180,E1 -22072.698,E2 -22072.698} C_VEL
LIN {X 0,Y 194.442,Z 599.815,A -85,B 0,C 180,E1 -22075.704,E2 -22075.704} C_VEL
LIN {X 0,Y 198.265,Z 592.674,A -85,B 0,C 180,E1 -22078.589,E2 -22078.589} C_VEL
LIN {X 0,Y 202.757,Z 583.828,A -85,B 0,C 180,E1 -22081.327,E2 -22081.327} C_VEL
LIN {X 0,Y 207.341,Z 573.793,A -85,B 0,C 180,E1 -22083.713,E2 -22083.713} C_VEL
LIN {X 0,Y 211.372,Z 563.566,A -85,B 0,C 180,E1 -22085.581,E2 -22085.581} C_VEL
LIN {X 0,Y 215.205,Z 552.258,A -85,B 0,C 180,E1 -22087.167,E2 -22087.167} C_VEL
LIN {X 0,Y 218.443,Z 540.545,A -85,B 0,C 180,E1 -22088.413,E2 -22088.413} C_VEL
LIN {X 0,Y 221.122,Z 527.733,A -85,B 0,C 180,E1 -22089.395,E2 -22089.395} C_VEL
LIN {X 0,Y 223.013,Z 514.867,A -85,B 0,C 180,E1 -22090.046,E2 -22090.046} C_VEL
LIN {X 0,Y 224.894,Z 486.889,A -85,B 0,C 180,E1 -22090.939,E2 -22090.939} C_VEL
LIN {X 0,Y 225.655,Z 473.399,A -85,B 0,C 180,E1 -22091.362,E2 -22091.362} C_VEL
LIN {X 0,Y 224.862,Z 467.049,A -85,B 0,C 180,E1 -22091.883,E2 -22091.883} C_VEL
LIN {X 0,Y 219.635,Z 454.713,A -85,B 0,C 180,E1 -22094.044,E2 -22094.044} C_VEL
LIN {X 0,Y 214.579,Z 444.362,A -85,B 0,C 180,E1 -22096.252,E2 -22096.252} C_VEL
LIN {X 0,Y 209.867,Z 435.858,A -85,B 0,C 180,E1 -22098.48,E2 -22098.48} C_VEL
LIN {X 0,Y 206.533,Z 430.207,A -85,B 0,C 180,E1 -22100.176,E2 -22100.176} C_VEL
LIN {X 0,Y 204.094,Z 426.188,A -85,B 0,C 180,E1 -22101.495,E2 -22101.495} C_VEL
LIN {X 0,Y 200.534,Z 420.685,A -85,B 0,C 180,E1 -22103.548,E2 -22103.548} C_VEL
LIN {X 0,Y 196.986,Z 415.397,A -85,B 0,C 180,E1 -22105.796,E2 -22105.796} C_VEL
LIN {X 0,Y 192.738,Z 409.722,A -85,B 0,C 180,E1 -22108.847,E2 -22108.847} C_VEL
LIN {X 0,Y 191.685,Z 408.112,A -85,B 0,C 180,E1 -22109.702,E2 -22109.702} C_VEL
LIN {X 0,Y 187.335,Z 402.635,A -85,B 0,C 180,E1 -22113.62,E2 -22113.62} C_VEL
LIN {X 0,Y 186.485,Z 401.049,A -85,B 0,C 180,E1 -22114.614,E2 -22114.614} C_VEL
LIN {X 0,Y 185.594,Z 398.355,A -85,B 0,C 180,E1 -22119.206,E2 -22119.206} C_VEL
LIN {X 0,Y 185.712,Z 398.337,A -85,B 0,C 180,E1 -22122.378,E2 -22122.378} C_VEL
LIN {X 0,Y 185.729,Z 398.335,A -85,B 0,C 180,E1 -22126.878,E2 -22126.878} C_VEL
LIN {X 0,Y 186.004,Z 398.303,A -85,B 0,C 180,E1 -22131.308,E2 -22131.308} C_VEL
LIN {X 0,Y 186.204,Z 398.273,A -85,B 0,C 180,E1 -22137.837,E2 -22137.837} C_VEL
LIN {X 0,Y 186.405,Z 398.267,A -85,B 0,C 180,E1 -22140.001,E2 -22140.001} C_VEL
LIN {X 0,Y 185.918,Z 398.32,A -85,B 0,C 180,E1 -22144.336,E2 -22144.336} C_VEL
LIN {X 0,Y 185.929,Z 398.32,A -85,B 0,C 180,E1 -22149.226,E2 -22149.226} C_VEL
LIN {X 0,Y 186.517,Z 400.467,A -85,B 0,C 180,E1 -22150.076,E2 -22150.076} C_VEL
LIN {X 0,Y 188.238,Z 402.878,A -85,B 0,C 180,E1 -22151.85,E2 -22151.85} C_VEL
LIN {X 0,Y 190.713,Z 404.38,A -85,B 0,C 180,E1 -22153.928,E2 -22153.928} C_VEL
LIN {X 0,Y 192.261,Z 407.35,A -85,B 0,C 180,E1 -22155.301,E2 -22155.301} C_VEL
LIN {X 0,Y 194.767,Z 409.583,A -85,B 0,C 180,E1 -22157.114,E2 -22157.114} C_VEL
LIN {X 0,Y 195.497,Z 410.503,A -85,B 0,C 180,E1 -22157.633,E2 -22157.633} C_VEL
LIN {X 0,Y 197.745,Z 413.74,A -85,B 0,C 180,E1 -22159.177,E2 -22159.177} C_VEL
LIN {X 0,Y 199.554,Z 415.531,A -85,B 0,C 180,E1 -22160.268,E2 -22160.268} C_VEL
LIN {X 0,Y 202.299,Z 419.239,A -85,B 0,C 180,E1 -22161.89,E2 -22161.89} C_VEL
LIN {X 0,Y 203.69,Z 421.043,A -85,B 0,C 180,E1 -22162.663,E2 -22162.663} C_VEL
LIN {X 0,Y 207.153,Z 425.784,A -85,B 0,C 180,E1 -22164.491,E2 -22164.491} C_VEL
LIN {X 0,Y 212.337,Z 433.1,A -85,B 0,C 180,E1 -22166.984,E2 -22166.984} C_VEL
LIN {X 0,Y 218.712,Z 443.014,A -85,B 0,C 180,E1 -22169.746,E2 -22169.746} C_VEL
LIN {X 0,Y 223.668,Z 451.848,A -85,B 0,C 180,E1 -22171.724,E2 -22171.724} C_VEL
LIN {X 0,Y 226.643,Z 458.262,A -85,B 0,C 180,E1 -22172.887,E2 -22172.887} C_VEL
LIN {X 0,Y 223.936,Z 499.036,A -85,B 0,C 180,E1 -22174.124,E2 -22174.124} C_VEL
